//     Enc/Inputs/In/nState1 @bit 4 <-> ENC Status compact/Status/Counter overflow
//     Enc/Inputs/In/nState1 @bit 3 <-> ENC Status compact/Status/Counter underflow
//     Enc/Inputs/In/nState1 @bit 7 <-> ENC Status compact/Status/Extrapolation stall
//     Enc/Inputs/In/nState1 <-> ENC Status compact/Status/Latch C valid
//     Enc/Inputs/In/nState1 @bit 1 <-> ENC Status compact/Status/Latch extern valid
//     Enc/Inputs/In/nState1 @bit 2 <-> ENC Status compact/Status/Set counter done
//     Enc/Inputs/In/nState2 @bit 4 <-> ENC Status compact/Status/Status of extern latch
//     Enc/Inputs/In/nState2 <-> ENC Status compact/Status/Status of input A
//     Enc/Inputs/In/nState2 @bit 1 <-> ENC Status compact/Status/Status of input B
//     Enc/Inputs/In/nState2 @bit 2 <-> ENC Status compact/Status/Status of input C
//     Enc/Inputs/In/nState2 @bit 5 <-> ENC Status compact/Status/Sync error
//     Enc/Inputs/In/nState2 @bit 7 <-> ENC Status compact/Status/TxPDO Toggle
//     Enc/Inputs/In/nState4 @bit 1 <-> WcState/InputToggle
//     Enc/Inputs/In/nState4 <-> WcState/WcState
//     Enc/Outputs/Out/nCtrl1 <-> ENC Control compact/Control/Enable latch C
//     Enc/Outputs/Out/nCtrl1 @bit 3 <-> ENC Control compact/Control/Enable latch extern on negative edge
//     Enc/Outputs/Out/nCtrl1 @bit 1 <-> ENC Control compact/Control/Enable latch extern on positive edge
//     Enc/Outputs/Out/nCtrl1 @bit 2 <-> ENC Control compact/Control/Set counter
//     Enc/Outputs/Out/nDataOut1[0] <-> ENC Control compact/Set counter value
//   NC-Task 1 SAF/Axes/NSH4 <-> Device 1 (EtherCAT)/Term 7 (EK1101)/Term 14 (EK1122)/Term 15 (EK1101)/NSH4 (N19) (EL7047)
//     Drive/Inputs/In/nState1 @bit 3 <-> STM Status/Status/Error
//     Drive/Inputs/In/nState1 @bit 7 <-> STM Status/Status/Motor stall
//     Drive/Inputs/In/nState1 @bit 5 <-> STM Status/Status/Moving negative
//     Drive/Inputs/In/nState1 @bit 4 <-> STM Status/Status/Moving positive
//     Drive/Inputs/In/nState1 @bit 1 <-> STM Status/Status/Ready
//     Drive/Inputs/In/nState1 <-> STM Status/Status/Ready to enable
//     Drive/Inputs/In/nState1 @bit 6 <-> STM Status/Status/Torque reduced
//     Drive/Inputs/In/nState1 @bit 2 <-> STM Status/Status/Warning
//     Drive/Inputs/In/nState2 @bit 3 <-> STM Status/Status/Digital input 1
//     Drive/Inputs/In/nState2 @bit 4 <-> STM Status/Status/Digital input 2
//     Drive/Inputs/In/nState2 @bit 5 <-> STM Status/Status/Sync error
//     Drive/Inputs/In/nState2 @bit 7 <-> STM Status/Status/TxPDO Toggle
//     Drive/Inputs/In/nState4 @bit 1 <-> WcState/InputToggle
//     Drive/Inputs/In/nState4 <-> WcState/WcState
//     Drive/Outputs/Out/nCtrl1 <-> STM Control/Control/Enable
//     Drive/Outputs/Out/nCtrl1 @bit 2 <-> STM Control/Control/Reduce torque
//     Drive/Outputs/Out/nCtrl1 @bit 1 <-> STM Control/Control/Reset
//     Drive/Outputs/Out/nCtrl2 @bit 3 <-> STM Control/Control/Digital output 1
//     Drive/Outputs/Out/nDataOut2[0] <-> STM Velocity/Velocity
//     Enc/Inputs/In/nDataIn1[0] <-> ENC Status compact/Counter value
//     Enc/Inputs/In/nDataIn2[0] <-> ENC Status compact/Latch value
//     Enc/Inputs/In/nState1 @bit 4 <-> ENC Status compact/Status/Counter overflow
//     Enc/Inputs/In/nState1 @bit 3 <-> ENC Status compact/Status/Counter underflow
//     Enc/Inputs/In/nState1 @bit 7 <-> ENC Status compact/Status/Extrapolation stall
//     Enc/Inputs/In/nState1 <-> ENC Status compact/Status/Latch C valid
//     Enc/Inputs/In/nState1 @bit 1 <-> ENC Status compact/Status/Latch extern valid
//     Enc/Inputs/In/nState1 @bit 2 <-> ENC Status compact/Status/Set counter done
//     Enc/Inputs/In/nState2 @bit 4 <-> ENC Status compact/Status/Status of extern latch
//     Enc/Inputs/In/nState2 <-> ENC Status compact/Status/Status of input A
//     Enc/Inputs/In/nState2 @bit 1 <-> ENC Status compact/Status/Status of input B
//     Enc/Inputs/In/nState2 @bit 2 <-> ENC Status compact/Status/Status of input C
//     Enc/Inputs/In/nState2 @bit 5 <-> ENC Status compact/Status/Sync error
//     Enc/Inputs/In/nState2 @bit 7 <-> ENC Status compact/Status/TxPDO Toggle
//     Enc/Inputs/In/nState4 @bit 1 <-> WcState/InputToggle
//     Enc/Inputs/In/nState4 <-> WcState/WcState
//     Enc/Outputs/Out/nCtrl1 <-> ENC Control compact/Control/Enable latch C
//     Enc/Outputs/Out/nCtrl1 @bit 3 <-> ENC Control compact/Control/Enable latch extern on negative edge
//     Enc/Outputs/Out/nCtrl1 @bit 1 <-> ENC Control compact/Control/Enable latch extern on positive edge
//     Enc/Outputs/Out/nCtrl1 @bit 2 <-> ENC Control compact/Control/Set counter
//     Enc/Outputs/Out/nDataOut1[0] <-> ENC Control compact/Set counter value
//   NC-Task 1 SAF/Axes/NTPA1 <-> Device 1 (EtherCAT)/Term 7 (EK1101)/Term 14 (EK1122)/Term 32 (EK1101)/NTPA1 - NTPA2 (N6) (EL7342)
//     Drive/Inputs/In/nState1 @bit 3 <-> DCM Status Channel 1/Status/Error
//     Drive/Inputs/In/nState1 @bit 5 <-> DCM Status Channel 1/Status/Moving negative
//     Drive/Inputs/In/nState1 @bit 4 <-> DCM Status Channel 1/Status/Moving positive
//     Drive/Inputs/In/nState1 @bit 1 <-> DCM Status Channel 1/Status/Ready
//     Drive/Inputs/In/nState1 <-> DCM Status Channel 1/Status/Ready to enable
//     Drive/Inputs/In/nState1 @bit 6 <-> DCM Status Channel 1/Status/Torque reduced
//     Drive/Inputs/In/nState1 @bit 2 <-> DCM Status Channel 1/Status/Warning
//     Drive/Inputs/In/nState2 @bit 3 <-> DCM Status Channel 1/Status/Digital input 1
//     Drive/Inputs/In/nState2 @bit 4 <-> DCM Status Channel 1/Status/Digital input 2
//     Drive/Inputs/In/nState2 @bit 5 <-> DCM Status Channel 1/Status/Sync error
//     Drive/Inputs/In/nState2 @bit 7 <-> DCM Status Channel 1/Status/TxPDO Toggle
//     Drive/Inputs/In/nState4 @bit 1 <-> WcState/InputToggle
//     Drive/Inputs/In/nState4 <-> WcState/WcState
//     Drive/Outputs/Out/nCtrl1 <-> DCM Control Channel 1/Control/Enable
//     Drive/Outputs/Out/nCtrl1 @bit 2 <-> DCM Control Channel 1/Control/Reduce torque
//     Drive/Outputs/Out/nCtrl1 @bit 1 <-> DCM Control Channel 1/Control/Reset
//     Drive/Outputs/Out/nCtrl1 @bit 3 <-> DCM Control Channel 1/Control/Threshold active
//     Drive/Outputs/Out/nDataOut2[0] <-> DCM Velocity Channel 1/Velocity
//     Enc/Inputs/In/nDataIn1[0] <-> ENC Status compact Channel 1/Counter value
//     Enc/Inputs/In/nDataIn2[0] <-> ENC Status compact Channel 1/Latch value
//     Enc/Inputs/In/nState1 @bit 4 <-> ENC Status compact Channel 1/Status/Counter overflow
//     Enc/Inputs/In/nState1 @bit 3 <-> ENC Status compact Channel 1/Status/Counter underflow
//     Enc/Inputs/In/nState1 @bit 7 <-> ENC Status compact Channel 1/Status/Extrapolation stall
//     Enc/Inputs/In/nState1 @bit 1 <-> ENC Status compact Channel 1/Status/Latch extern valid
//     Enc/Inputs/In/nState1 @bit 2 <-> ENC Status compact Channel 1/Status/Set counter done
//     Enc/Inputs/In/nState2 @bit 4 <-> ENC Status compact Channel 1/Status/Status of extern latch
//     Enc/Inputs/In/nState2 <-> ENC Status compact Channel 1/Status/Status of input A
//     Enc/Inputs/In/nState2 @bit 1 <-> ENC Status compact Channel 1/Status/Status of input B
//     Enc/Inputs/In/nState2 @bit 5 <-> ENC Status compact Channel 1/Status/Sync error
//     Enc/Inputs/In/nState2 @bit 7 <-> ENC Status compact Channel 1/Status/TxPDO Toggle
//     Enc/Inputs/In/nState4 @bit 1 <-> WcState/InputToggle
//     Enc/Inputs/In/nState4 <-> WcState/WcState
//     Enc/Outputs/Out/nCtrl1 @bit 3 <-> ENC Control compact Channel 1/Control/Enable latch extern on negative edge
//     Enc/Outputs/Out/nCtrl1 @bit 1 <-> ENC Control compact Channel 1/Control/Enable latch extern on positive edge
//     Enc/Outputs/Out/nCtrl1 @bit 2 <-> ENC Control compact Channel 1/Control/Set counter
//     Enc/Outputs/Out/nDataOut1[0] <-> ENC Control compact Channel 1/Set counter value
//   NC-Task 1 SAF/Axes/NTPA2 <-> Device 1 (EtherCAT)/Term 7 (EK1101)/Term 14 (EK1122)/Term 32 (EK1101)/NTPA1 - NTPA2 (N6) (EL7342)
//     Drive/Inputs/In/nState1 @bit 3 <-> DCM Status Channel 2/Status/Error
//     Drive/Inputs/In/nState1 @bit 5 <-> DCM Status Channel 2/Status/Moving negative
//     Drive/Inputs/In/nState1 @bit 4 <-> DCM Status Channel 2/Status/Moving positive
//     Drive/Inputs/In/nState1 @bit 1 <-> DCM Status Channel 2/Status/Ready
//     Drive/Inputs/In/nState1 <-> DCM Status Channel 2/Status/Ready to enable
//     Drive/Inputs/In/nState1 @bit 6 <-> DCM Status Channel 2/Status/Torque reduced
//     Drive/Inputs/In/nState1 @bit 2 <-> DCM Status Channel 2/Status/Warning
//     Drive/Inputs/In/nState2 @bit 3 <-> DCM Status Channel 2/Status/Digital input 1
//     Drive/Inputs/In/nState2 @bit 4 <-> DCM Status Channel 2/Status/Digital input 2
//     Drive/Inputs/In/nState2 @bit 5 <-> DCM Status Channel 2/Status/Sync error
//     Drive/Inputs/In/nState2 @bit 7 <-> DCM Status Channel 2/Status/TxPDO Toggle
//     Drive/Inputs/In/nState4 @bit 1 <-> WcState/InputToggle
//     Drive/Inputs/In/nState4 <-> WcState/WcState
//     Drive/Outputs/Out/nCtrl1 <-> DCM Control Channel 2/Control/Enable
//     Drive/Outputs/Out/nCtrl1 @bit 2 <-> DCM Control Channel 2/Control/Reduce torque
//     Drive/Outputs/Out/nCtrl1 @bit 1 <-> DCM Control Channel 2/Control/Reset
//     Drive/Outputs/Out/nCtrl1 @bit 3 <-> DCM Control Channel 2/Control/Threshold active
//     Drive/Outputs/Out/nDataOut2[0] <-> DCM Velocity Channel 2/Velocity
//     Enc/Inputs/In/nDataIn1[0] <-> ENC Status compact Channel 2/Counter value
//     Enc/Inputs/In/nDataIn2[0] <-> ENC Status compact Channel 2/Latch value
//     Enc/Inputs/In/nState1 @bit 4 <-> ENC Status compact Channel 2/Status/Counter overflow
//     Enc/Inputs/In/nState1 @bit 3 <-> ENC Status compact Channel 2/Status/Counter underflow
//     Enc/Inputs/In/nState1 @bit 7 <-> ENC Status compact Channel 2/Status/Extrapolation stall
//     Enc/Inputs/In/nState1 @bit 1 <-> ENC Status compact Channel 2/Status/Latch extern valid
//     Enc/Inputs/In/nState1 @bit 2 <-> ENC Status compact Channel 2/Status/Set counter done
//     Enc/Inputs/In/nState2 @bit 4 <-> ENC Status compact Channel 2/Status/Status of extern latch
//     Enc/Inputs/In/nState2 <-> ENC Status compact Channel 2/Status/Status of input A
//     Enc/Inputs/In/nState2 @bit 1 <-> ENC Status compact Channel 2/Status/Status of input B
//     Enc/Inputs/In/nState2 @bit 5 <-> ENC Status compact Channel 2/Status/Sync error
//     Enc/Inputs/In/nState2 @bit 7 <-> ENC Status compact Channel 2/Status/TxPDO Toggle
//     Enc/Inputs/In/nState4 @bit 1 <-> WcState/InputToggle
//     Enc/Inputs/In/nState4 <-> WcState/WcState
//     Enc/Outputs/Out/nCtrl1 @bit 3 <-> ENC Control compact Channel 2/Control/Enable latch extern on negative edge
//     Enc/Outputs/Out/nCtrl1 @bit 1 <-> ENC Control compact Channel 2/Control/Enable latch extern on positive edge
//     Enc/Outputs/Out/nCtrl1 @bit 2 <-> ENC Control compact Channel 2/Control/Set counter
//     Enc/Outputs/Out/nDataOut1[0] <-> ENC Control compact Channel 2/Set counter value
//   NC-Task 1 SAF/Axes/NTPA3 <-> Device 1 (EtherCAT)/Term 7 (EK1101)/Term 14 (EK1122)/Term 32 (EK1101)/NTPA3 - NTPA4 (N7) (EL7342)
//     Drive/Inputs/In/nState1 @bit 3 <-> DCM Status Channel 1/Status/Error
//     Drive/Inputs/In/nState1 @bit 5 <-> DCM Status Channel 1/Status/Moving negative
//     Drive/Inputs/In/nState1 @bit 4 <-> DCM Status Channel 1/Status/Moving positive
//     Drive/Inputs/In/nState1 @bit 1 <-> DCM Status Channel 1/Status/Ready
//     Drive/Inputs/In/nState1 <-> DCM Status Channel 1/Status/Ready to enable
//     Drive/Inputs/In/nState1 @bit 6 <-> DCM Status Channel 1/Status/Torque reduced
//     Drive/Inputs/In/nState1 @bit 2 <-> DCM Status Channel 1/Status/Warning
//     Drive/Inputs/In/nState2 @bit 3 <-> DCM Status Channel 1/Status/Digital input 1
//     Drive/Inputs/In/nState2 @bit 4 <-> DCM Status Channel 1/Status/Digital input 2
//     Drive/Inputs/In/nState2 @bit 5 <-> DCM Status Channel 1/Status/Sync error
//     Drive/Inputs/In/nState2 @bit 7 <-> DCM Status Channel 1/Status/TxPDO Toggle
//     Drive/Inputs/In/nState4 @bit 1 <-> WcState/InputToggle
//     Drive/Inputs/In/nState4 <-> WcState/WcState
//     Drive/Outputs/Out/nCtrl1 <-> DCM Control Channel 1/Control/Enable
//     Drive/Outputs/Out/nCtrl1 @bit 2 <-> DCM Control Channel 1/Control/Reduce torque
//     Drive/Outputs/Out/nCtrl1 @bit 1 <-> DCM Control Channel 1/Control/Reset
//     Drive/Outputs/Out/nCtrl1 @bit 3 <-> DCM Control Channel 1/Control/Threshold active
//     Drive/Outputs/Out/nDataOut2[0] <-> DCM Velocity Channel 1/Velocity
//     Enc/Inputs/In/nDataIn1[0] <-> ENC Status compact Channel 1/Counter value
//     Enc/Inputs/In/nDataIn2[0] <-> ENC Status compact Channel 1/Latch value
//     Enc/Inputs/In/nState1 @bit 4 <-> ENC Status compact Channel 1/Status/Counter overflow
//     Enc/Inputs/In/nState1 @bit 3 <-> ENC Status compact Channel 1/Status/Counter underflow
//     Enc/Inputs/In/nState1 @bit 7 <-> ENC Status compact Channel 1/Status/Extrapolation stall
//     Enc/Inputs/In/nState1 @bit 1 <-> ENC Status compact Channel 1/Status/Latch extern valid
//     Enc/Inputs/In/nState1 @bit 2 <-> ENC Status compact Channel 1/Status/Set counter done
//     Enc/Inputs/In/nState2 @bit 4 <-> ENC Status compact Channel 1/Status/Status of extern latch
//     Enc/Inputs/In/nState2 <-> ENC Status compact Channel 1/Status/Status of input A
//     Enc/Inputs/In/nState2 @bit 1 <-> ENC Status compact Channel 1/Status/Status of input B
//     Enc/Inputs/In/nState2 @bit 5 <-> ENC Status compact Channel 1/Status/Sync error
//     Enc/Inputs/In/nState2 @bit 7 <-> ENC Status compact Channel 1/Status/TxPDO Toggle
//     Enc/Inputs/In/nState4 @bit 1 <-> WcState/InputToggle
//     Enc/Inputs/In/nState4 <-> WcState/WcState
//     Enc/Outputs/Out/nCtrl1 @bit 3 <-> ENC Control compact Channel 1/Control/Enable latch extern on negative edge
//     Enc/Outputs/Out/nCtrl1 @bit 1 <-> ENC Control compact Channel 1/Control/Enable latch extern on positive edge
//     Enc/Outputs/Out/nCtrl1 @bit 2 <-> ENC Control compact Channel 1/Control/Set counter
//     Enc/Outputs/Out/nDataOut1[0] <-> ENC Control compact Channel 1/Set counter value
//   NC-Task 1 SAF/Axes/NTPA4 <-> Device 1 (EtherCAT)/Term 7 (EK1101)/Term 14 (EK1122)/Term 32 (EK1101)/NTPA3 - NTPA4 (N7) (EL7342)
//     Drive/Inputs/In/nState1 @bit 3 <-> DCM Status Channel 2/Status/Error
//     Drive/Inputs/In/nState1 @bit 5 <-> DCM Status Channel 2/Status/Moving negative
//     Drive/Inputs/In/nState1 @bit 4 <-> DCM Status Channel 2/Status/Moving positive
//     Drive/Inputs/In/nState1 @bit 1 <-> DCM Status Channel 2/Status/Ready
//     Drive/Inputs/In/nState1 <-> DCM Status Channel 2/Status/Ready to enable
//     Drive/Inputs/In/nState1 @bit 6 <-> DCM Status Channel 2/Status/Torque reduced
//     Drive/Inputs/In/nState1 @bit 2 <-> DCM Status Channel 2/Status/Warning
//     Drive/Inputs/In/nState2 @bit 3 <-> DCM Status Channel 2/Status/Digital input 1
//     Drive/Inputs/In/nState2 @bit 4 <-> DCM Status Channel 2/Status/Digital input 2
//     Drive/Inputs/In/nState2 @bit 5 <-> DCM Status Channel 2/Status/Sync error
//     Drive/Inputs/In/nState2 @bit 7 <-> DCM Status Channel 2/Status/TxPDO Toggle
//     Drive/Inputs/In/nState4 @bit 1 <-> WcState/InputToggle
//     Drive/Inputs/In/nState4 <-> WcState/WcState
//     Drive/Outputs/Out/nCtrl1 <-> DCM Control Channel 2/Control/Enable
//     Drive/Outputs/Out/nCtrl1 @bit 2 <-> DCM Control Channel 2/Control/Reduce torque
//     Drive/Outputs/Out/nCtrl1 @bit 1 <-> DCM Control Channel 2/Control/Reset
//     Drive/Outputs/Out/nCtrl1 @bit 3 <-> DCM Control Channel 2/Control/Threshold active
//     Drive/Outputs/Out/nDataOut2[0] <-> DCM Velocity Channel 2/Velocity
//     Enc/Inputs/In/nDataIn1[0] <-> ENC Status compact Channel 2/Counter value
//     Enc/Inputs/In/nDataIn2[0] <-> ENC Status compact Channel 2/Latch value
//     Enc/Inputs/In/nState1 @bit 4 <-> ENC Status compact Channel 2/Status/Counter overflow
//     Enc/Inputs/In/nState1 @bit 3 <-> ENC Status compact Channel 2/Status/Counter underflow
//     Enc/Inputs/In/nState1 @bit 7 <-> ENC Status compact Channel 2/Status/Extrapolation stall
//     Enc/Inputs/In/nState1 @bit 1 <-> ENC Status compact Channel 2/Status/Latch extern valid
//     Enc/Inputs/In/nState1 @bit 2 <-> ENC Status compact Channel 2/Status/Set counter done
//     Enc/Inputs/In/nState2 @bit 4 <-> ENC Status compact Channel 2/Status/Status of extern latch
//     Enc/Inputs/In/nState2 <-> ENC Status compact Channel 2/Status/Status of input A
//     Enc/Inputs/In/nState2 @bit 1 <-> ENC Status compact Channel 2/Status/Status of input B
//     Enc/Inputs/In/nState2 @bit 5 <-> ENC Status compact Channel 2/Status/Sync error
//     Enc/Inputs/In/nState2 @bit 7 <-> ENC Status compact Channel 2/Status/TxPDO Toggle
//     Enc/Inputs/In/nState4 @bit 1 <-> WcState/InputToggle
//     Enc/Inputs/In/nState4 <-> WcState/WcState
//     Enc/Outputs/Out/nCtrl1 @bit 3 <-> ENC Control compact Channel 2/Control/Enable latch extern on negative edge
//     Enc/Outputs/Out/nCtrl1 @bit 1 <-> ENC Control compact Channel 2/Control/Enable latch extern on positive edge
//     Enc/Outputs/Out/nCtrl1 @bit 2 <-> ENC Control compact Channel 2/Control/Set counter
//     Enc/Outputs/Out/nDataOut1[0] <-> ENC Control compact Channel 2/Set counter value
//   NC-Task 1 SAF/Axes/NTPB1 <-> Device 1 (EtherCAT)/Term 7 (EK1101)/Term 14 (EK1122)/Term 32 (EK1101)/NTPB1 - NTPB2 (N14) (EL7342)
//     Drive/Inputs/In/nState1 @bit 3 <-> DCM Status Channel 1/Status/Error
//     Drive/Inputs/In/nState1 @bit 5 <-> DCM Status Channel 1/Status/Moving negative
//     Drive/Inputs/In/nState1 @bit 4 <-> DCM Status Channel 1/Status/Moving positive
//     Drive/Inputs/In/nState1 @bit 1 <-> DCM Status Channel 1/Status/Ready
//     Drive/Inputs/In/nState1 <-> DCM Status Channel 1/Status/Ready to enable
//     Drive/Inputs/In/nState1 @bit 6 <-> DCM Status Channel 1/Status/Torque reduced
//     Drive/Inputs/In/nState1 @bit 2 <-> DCM Status Channel 1/Status/Warning
//     Drive/Inputs/In/nState2 @bit 3 <-> DCM Status Channel 1/Status/Digital input 1
//     Drive/Inputs/In/nState2 @bit 4 <-> DCM Status Channel 1/Status/Digital input 2
//     Drive/Inputs/In/nState2 @bit 5 <-> DCM Status Channel 1/Status/Sync error
//     Drive/Inputs/In/nState2 @bit 7 <-> DCM Status Channel 1/Status/TxPDO Toggle
//     Drive/Inputs/In/nState4 @bit 1 <-> WcState/InputToggle
//     Drive/Inputs/In/nState4 <-> WcState/WcState
//     Drive/Outputs/Out/nCtrl1 <-> DCM Control Channel 1/Control/Enable
//     Drive/Outputs/Out/nCtrl1 @bit 2 <-> DCM Control Channel 1/Control/Reduce torque
//     Drive/Outputs/Out/nCtrl1 @bit 1 <-> DCM Control Channel 1/Control/Reset
//     Drive/Outputs/Out/nCtrl1 @bit 3 <-> DCM Control Channel 1/Control/Threshold active
//     Drive/Outputs/Out/nDataOut2[0] <-> DCM Velocity Channel 1/Velocity
//     Enc/Inputs/In/nDataIn1[0] <-> ENC Status compact Channel 1/Counter value
//     Enc/Inputs/In/nDataIn2[0] <-> ENC Status compact Channel 1/Latch value
//     Enc/Inputs/In/nState1 @bit 4 <-> ENC Status compact Channel 1/Status/Counter overflow
//     Enc/Inputs/In/nState1 @bit 3 <-> ENC Status compact Channel 1/Status/Counter underflow
//     Enc/Inputs/In/nState1 @bit 7 <-> ENC Status compact Channel 1/Status/Extrapolation stall
//     Enc/Inputs/In/nState1 @bit 1 <-> ENC Status compact Channel 1/Status/Latch extern valid
//     Enc/Inputs/In/nState1 @bit 2 <-> ENC Status compact Channel 1/Status/Set counter done
//     Enc/Inputs/In/nState2 @bit 4 <-> ENC Status compact Channel 1/Status/Status of extern latch
//     Enc/Inputs/In/nState2 <-> ENC Status compact Channel 1/Status/Status of input A
//     Enc/Inputs/In/nState2 @bit 1 <-> ENC Status compact Channel 1/Status/Status of input B
//     Enc/Inputs/In/nState2 @bit 5 <-> ENC Status compact Channel 1/Status/Sync error
//     Enc/Inputs/In/nState2 @bit 7 <-> ENC Status compact Channel 1/Status/TxPDO Toggle
//     Enc/Inputs/In/nState4 @bit 1 <-> WcState/InputToggle
//     Enc/Inputs/In/nState4 <-> WcState/WcState
//     Enc/Outputs/Out/nCtrl1 @bit 3 <-> ENC Control compact Channel 1/Control/Enable latch extern on negative edge
//     Enc/Outputs/Out/nCtrl1 @bit 1 <-> ENC Control compact Channel 1/Control/Enable latch extern on positive edge
//     Enc/Outputs/Out/nCtrl1 @bit 2 <-> ENC Control compact Channel 1/Control/Set counter
//     Enc/Outputs/Out/nDataOut1[0] <-> ENC Control compact Channel 1/Set counter value
//   NC-Task 1 SAF/Axes/NTPB2 <-> Device 1 (EtherCAT)/Term 7 (EK1101)/Term 14 (EK1122)/Term 32 (EK1101)/NTPB1 - NTPB2 (N14) (EL7342)
//     Drive/Inputs/In/nState1 @bit 3 <-> DCM Status Channel 2/Status/Error
//     Drive/Inputs/In/nState1 @bit 5 <-> DCM Status Channel 2/Status/Moving negative
//     Drive/Inputs/In/nState1 @bit 4 <-> DCM Status Channel 2/Status/Moving positive
//     Drive/Inputs/In/nState1 @bit 1 <-> DCM Status Channel 2/Status/Ready
//     Drive/Inputs/In/nState1 <-> DCM Status Channel 2/Status/Ready to enable
//     Drive/Inputs/In/nState1 @bit 6 <-> DCM Status Channel 2/Status/Torque reduced
//     Drive/Inputs/In/nState1 @bit 2 <-> DCM Status Channel 2/Status/Warning
//     Drive/Inputs/In/nState2 @bit 3 <-> DCM Status Channel 2/Status/Digital input 1
//     Drive/Inputs/In/nState2 @bit 4 <-> DCM Status Channel 2/Status/Digital input 2
//     Drive/Inputs/In/nState2 @bit 5 <-> DCM Status Channel 2/Status/Sync error
//     Drive/Inputs/In/nState2 @bit 7 <-> DCM Status Channel 2/Status/TxPDO Toggle
//     Drive/Inputs/In/nState4 @bit 1 <-> WcState/InputToggle
//     Drive/Inputs/In/nState4 <-> WcState/WcState
//     Drive/Outputs/Out/nCtrl1 <-> DCM Control Channel 2/Control/Enable
//     Drive/Outputs/Out/nCtrl1 @bit 2 <-> DCM Control Channel 2/Control/Reduce torque
//     Drive/Outputs/Out/nCtrl1 @bit 1 <-> DCM Control Channel 2/Control/Reset
//     Drive/Outputs/Out/nCtrl1 @bit 3 <-> DCM Control Channel 2/Control/Threshold active
//     Drive/Outputs/Out/nDataOut2[0] <-> DCM Velocity Channel 2/Velocity
//     Enc/Inputs/In/nDataIn1[0] <-> ENC Status compact Channel 2/Counter value
//     Enc/Inputs/In/nDataIn2[0] <-> ENC Status compact Channel 2/Latch value
//     Enc/Inputs/In/nState1 @bit 4 <-> ENC Status compact Channel 2/Status/Counter overflow
//     Enc/Inputs/In/nState1 @bit 3 <-> ENC Status compact Channel 2/Status/Counter underflow
//     Enc/Inputs/In/nState1 @bit 7 <-> ENC Status compact Channel 2/Status/Extrapolation stall
//     Enc/Inputs/In/nState1 @bit 1 <-> ENC Status compact Channel 2/Status/Latch extern valid
//     Enc/Inputs/In/nState1 @bit 2 <-> ENC Status compact Channel 2/Status/Set counter done
//     Enc/Inputs/In/nState2 @bit 4 <-> ENC Status compact Channel 2/Status/Status of extern latch
//     Enc/Inputs/In/nState2 <-> ENC Status compact Channel 2/Status/Status of input A
//     Enc/Inputs/In/nState2 @bit 1 <-> ENC Status compact Channel 2/Status/Status of input B
//     Enc/Inputs/In/nState2 @bit 5 <-> ENC Status compact Channel 2/Status/Sync error
//     Enc/Inputs/In/nState2 @bit 7 <-> ENC Status compact Channel 2/Status/TxPDO Toggle
//     Enc/Inputs/In/nState4 @bit 1 <-> WcState/InputToggle
//     Enc/Inputs/In/nState4 <-> WcState/WcState
//     Enc/Outputs/Out/nCtrl1 @bit 3 <-> ENC Control compact Channel 2/Control/Enable latch extern on negative edge
//     Enc/Outputs/Out/nCtrl1 @bit 1 <-> ENC Control compact Channel 2/Control/Enable latch extern on positive edge
//     Enc/Outputs/Out/nCtrl1 @bit 2 <-> ENC Control compact Channel 2/Control/Set counter
//     Enc/Outputs/Out/nDataOut1[0] <-> ENC Control compact Channel 2/Set counter value
//   NC-Task 1 SAF/Axes/NTPB3 <-> Device 1 (EtherCAT)/Term 7 (EK1101)/Term 14 (EK1122)/Term 32 (EK1101)/NTPB3 - NTPB4 (N15) (EL7342)
//     Drive/Inputs/In/nState1 @bit 3 <-> DCM Status Channel 1/Status/Error
//     Drive/Inputs/In/nState1 @bit 5 <-> DCM Status Channel 1/Status/Moving negative
//     Drive/Inputs/In/nState1 @bit 4 <-> DCM Status Channel 1/Status/Moving positive
//     Drive/Inputs/In/nState1 @bit 1 <-> DCM Status Channel 1/Status/Ready
//     Drive/Inputs/In/nState1 <-> DCM Status Channel 1/Status/Ready to enable
//     Drive/Inputs/In/nState1 @bit 6 <-> DCM Status Channel 1/Status/Torque reduced
//     Drive/Inputs/In/nState1 @bit 2 <-> DCM Status Channel 1/Status/Warning
//     Drive/Inputs/In/nState2 @bit 3 <-> DCM Status Channel 1/Status/Digital input 1
//     Drive/Inputs/In/nState2 @bit 4 <-> DCM Status Channel 1/Status/Digital input 2
//     Drive/Inputs/In/nState2 @bit 5 <-> DCM Status Channel 1/Status/Sync error
//     Drive/Inputs/In/nState2 @bit 7 <-> DCM Status Channel 1/Status/TxPDO Toggle
//     Drive/Inputs/In/nState4 @bit 1 <-> WcState/InputToggle
//     Drive/Inputs/In/nState4 <-> WcState/WcState
//     Drive/Outputs/Out/nCtrl1 <-> DCM Control Channel 1/Control/Enable
//     Drive/Outputs/Out/nCtrl1 @bit 2 <-> DCM Control Channel 1/Control/Reduce torque
//     Drive/Outputs/Out/nCtrl1 @bit 1 <-> DCM Control Channel 1/Control/Reset
//     Drive/Outputs/Out/nCtrl1 @bit 3 <-> DCM Control Channel 1/Control/Threshold active
//     Drive/Outputs/Out/nDataOut2[0] <-> DCM Velocity Channel 1/Velocity
//     Enc/Inputs/In/nDataIn1[0] <-> ENC Status compact Channel 1/Counter value
//     Enc/Inputs/In/nDataIn2[0] <-> ENC Status compact Channel 1/Latch value
//     Enc/Inputs/In/nState1 @bit 4 <-> ENC Status compact Channel 1/Status/Counter overflow
//     Enc/Inputs/In/nState1 @bit 3 <-> ENC Status compact Channel 1/Status/Counter underflow
//     Enc/Inputs/In/nState1 @bit 7 <-> ENC Status compact Channel 1/Status/Extrapolation stall
//     Enc/Inputs/In/nState1 @bit 1 <-> ENC Status compact Channel 1/Status/Latch extern valid
//     Enc/Inputs/In/nState1 @bit 2 <-> ENC Status compact Channel 1/Status/Set counter done
//     Enc/Inputs/In/nState2 @bit 4 <-> ENC Status compact Channel 1/Status/Status of extern latch
//     Enc/Inputs/In/nState2 <-> ENC Status compact Channel 1/Status/Status of input A
//     Enc/Inputs/In/nState2 @bit 1 <-> ENC Status compact Channel 1/Status/Status of input B
//     Enc/Inputs/In/nState2 @bit 5 <-> ENC Status compact Channel 1/Status/Sync error
//     Enc/Inputs/In/nState2 @bit 7 <-> ENC Status compact Channel 1/Status/TxPDO Toggle
//     Enc/Inputs/In/nState4 @bit 1 <-> WcState/InputToggle
//     Enc/Inputs/In/nState4 <-> WcState/WcState
//     Enc/Outputs/Out/nCtrl1 @bit 3 <-> ENC Control compact Channel 1/Control/Enable latch extern on negative edge
//     Enc/Outputs/Out/nCtrl1 @bit 1 <-> ENC Control compact Channel 1/Control/Enable latch extern on positive edge
//     Enc/Outputs/Out/nCtrl1 @bit 2 <-> ENC Control compact Channel 1/Control/Set counter
//     Enc/Outputs/Out/nDataOut1[0] <-> ENC Control compact Channel 1/Set counter value
//   NC-Task 1 SAF/Axes/NTPB4 <-> Device 1 (EtherCAT)/Term 7 (EK1101)/Term 14 (EK1122)/Term 32 (EK1101)/NTPB3 - NTPB4 (N15) (EL7342)
//     Drive/Inputs/In/nState1 @bit 3 <-> DCM Status Channel 2/Status/Error
//     Drive/Inputs/In/nState1 @bit 5 <-> DCM Status Channel 2/Status/Moving negative
//     Drive/Inputs/In/nState1 @bit 4 <-> DCM Status Channel 2/Status/Moving positive
//     Drive/Inputs/In/nState1 @bit 1 <-> DCM Status Channel 2/Status/Ready
//     Drive/Inputs/In/nState1 <-> DCM Status Channel 2/Status/Ready to enable
//     Drive/Inputs/In/nState1 @bit 6 <-> DCM Status Channel 2/Status/Torque reduced
//     Drive/Inputs/In/nState1 @bit 2 <-> DCM Status Channel 2/Status/Warning
//     Drive/Inputs/In/nState2 @bit 3 <-> DCM Status Channel 2/Status/Digital input 1
//     Drive/Inputs/In/nState2 @bit 4 <-> DCM Status Channel 2/Status/Digital input 2
//     Drive/Inputs/In/nState2 @bit 5 <-> DCM Status Channel 2/Status/Sync error
//     Drive/Inputs/In/nState2 @bit 7 <-> DCM Status Channel 2/Status/TxPDO Toggle
//     Drive/Inputs/In/nState4 @bit 1 <-> WcState/InputToggle
//     Drive/Inputs/In/nState4 <-> WcState/WcState
//     Drive/Outputs/Out/nCtrl1 <-> DCM Control Channel 2/Control/Enable
//     Drive/Outputs/Out/nCtrl1 @bit 2 <-> DCM Control Channel 2/Control/Reduce torque
//     Drive/Outputs/Out/nCtrl1 @bit 1 <-> DCM Control Channel 2/Control/Reset
//     Drive/Outputs/Out/nCtrl1 @bit 3 <-> DCM Control Channel 2/Control/Threshold active
//     Drive/Outputs/Out/nDataOut2[0] <-> DCM Velocity Channel 2/Velocity
//     Enc/Inputs/In/nDataIn1[0] <-> ENC Status compact Channel 2/Counter value
//     Enc/Inputs/In/nDataIn2[0] <-> ENC Status compact Channel 2/Latch value
//     Enc/Inputs/In/nState1 @bit 4 <-> ENC Status compact Channel 2/Status/Counter overflow
//     Enc/Inputs/In/nState1 @bit 3 <-> ENC Status compact Channel 2/Status/Counter underflow
//     Enc/Inputs/In/nState1 @bit 7 <-> ENC Status compact Channel 2/Status/Extrapolation stall
//     Enc/Inputs/In/nState1 @bit 1 <-> ENC Status compact Channel 2/Status/Latch extern valid
//     Enc/Inputs/In/nState1 @bit 2 <-> ENC Status compact Channel 2/Status/Set counter done
//     Enc/Inputs/In/nState2 @bit 4 <-> ENC Status compact Channel 2/Status/Status of extern latch
//     Enc/Inputs/In/nState2 <-> ENC Status compact Channel 2/Status/Status of input A
//     Enc/Inputs/In/nState2 @bit 1 <-> ENC Status compact Channel 2/Status/Status of input B
//     Enc/Inputs/In/nState2 @bit 5 <-> ENC Status compact Channel 2/Status/Sync error
//     Enc/Inputs/In/nState2 @bit 7 <-> ENC Status compact Channel 2/Status/TxPDO Toggle
//     Enc/Inputs/In/nState4 @bit 1 <-> WcState/InputToggle
//     Enc/Inputs/In/nState4 <-> WcState/WcState
//     Enc/Outputs/Out/nCtrl1 @bit 3 <-> ENC Control compact Channel 2/Control/Enable latch extern on negative edge
//     Enc/Outputs/Out/nCtrl1 @bit 1 <-> ENC Control compact Channel 2/Control/Enable latch extern on positive edge
//     Enc/Outputs/Out/nCtrl1 @bit 2 <-> ENC Control compact Channel 2/Control/Set counter
//     Enc/Outputs/Out/nDataOut1[0] <-> ENC Control compact Channel 2/Set counter value
//   NC-Task 1 SAF/Axes/NTTA1 <-> Device 1 (EtherCAT)/Term 7 (EK1101)/Term 14 (EK1122)/Term 32 (EK1101)/NTTA1 - NTTA2 (N9) (EL7342)
//     Drive/Inputs/In/nState1 @bit 3 <-> DCM Status Channel 1/Status/Error
//     Drive/Inputs/In/nState1 @bit 5 <-> DCM Status Channel 1/Status/Moving negative
//     Drive/Inputs/In/nState1 @bit 4 <-> DCM Status Channel 1/Status/Moving positive
//     Drive/Inputs/In/nState1 @bit 1 <-> DCM Status Channel 1/Status/Ready
//     Drive/Inputs/In/nState1 <-> DCM Status Channel 1/Status/Ready to enable
//     Drive/Inputs/In/nState1 @bit 6 <-> DCM Status Channel 1/Status/Torque reduced
//     Drive/Inputs/In/nState1 @bit 2 <-> DCM Status Channel 1/Status/Warning
//     Drive/Inputs/In/nState2 @bit 3 <-> DCM Status Channel 1/Status/Digital input 1
//     Drive/Inputs/In/nState2 @bit 4 <-> DCM Status Channel 1/Status/Digital input 2
//     Drive/Inputs/In/nState2 @bit 5 <-> DCM Status Channel 1/Status/Sync error
//     Drive/Inputs/In/nState2 @bit 7 <-> DCM Status Channel 1/Status/TxPDO Toggle
//     Drive/Inputs/In/nState4 @bit 1 <-> WcState/InputToggle
//     Drive/Inputs/In/nState4 <-> WcState/WcState
//     Drive/Outputs/Out/nCtrl1 <-> DCM Control Channel 1/Control/Enable
//     Drive/Outputs/Out/nCtrl1 @bit 2 <-> DCM Control Channel 1/Control/Reduce torque
//     Drive/Outputs/Out/nCtrl1 @bit 1 <-> DCM Control Channel 1/Control/Reset
//     Drive/Outputs/Out/nCtrl1 @bit 3 <-> DCM Control Channel 1/Control/Threshold active
//     Drive/Outputs/Out/nDataOut2[0] <-> DCM Velocity Channel 1/Velocity
//     Enc/Inputs/In/nDataIn1[0] <-> ENC Status compact Channel 1/Counter value
//     Enc/Inputs/In/nDataIn2[0] <-> ENC Status compact Channel 1/Latch value
//     Enc/Inputs/In/nState1 @bit 4 <-> ENC Status compact Channel 1/Status/Counter overflow
//     Enc/Inputs/In/nState1 @bit 3 <-> ENC Status compact Channel 1/Status/Counter underflow
//     Enc/Inputs/In/nState1 @bit 7 <-> ENC Status compact Channel 1/Status/Extrapolation stall
//     Enc/Inputs/In/nState1 @bit 1 <-> ENC Status compact Channel 1/Status/Latch extern valid
//     Enc/Inputs/In/nState1 @bit 2 <-> ENC Status compact Channel 1/Status/Set counter done
//     Enc/Inputs/In/nState2 @bit 4 <-> ENC Status compact Channel 1/Status/Status of extern latch
//     Enc/Inputs/In/nState2 <-> ENC Status compact Channel 1/Status/Status of input A
//     Enc/Inputs/In/nState2 @bit 1 <-> ENC Status compact Channel 1/Status/Status of input B
//     Enc/Inputs/In/nState2 @bit 5 <-> ENC Status compact Channel 1/Status/Sync error
//     Enc/Inputs/In/nState2 @bit 7 <-> ENC Status compact Channel 1/Status/TxPDO Toggle
//     Enc/Inputs/In/nState4 @bit 1 <-> WcState/InputToggle
//     Enc/Inputs/In/nState4 <-> WcState/WcState
//     Enc/Outputs/Out/nCtrl1 @bit 3 <-> ENC Control compact Channel 1/Control/Enable latch extern on negative edge
//     Enc/Outputs/Out/nCtrl1 @bit 1 <-> ENC Control compact Channel 1/Control/Enable latch extern on positive edge
//     Enc/Outputs/Out/nCtrl1 @bit 2 <-> ENC Control compact Channel 1/Control/Set counter
//     Enc/Outputs/Out/nDataOut1[0] <-> ENC Control compact Channel 1/Set counter value
//   NC-Task 1 SAF/Axes/NTTA2 <-> Device 1 (EtherCAT)/Term 7 (EK1101)/Term 14 (EK1122)/Term 32 (EK1101)/NTTA1 - NTTA2 (N9) (EL7342)
//     Drive/Inputs/In/nState1 @bit 3 <-> DCM Status Channel 2/Status/Error
//     Drive/Inputs/In/nState1 @bit 5 <-> DCM Status Channel 2/Status/Moving negative
//     Drive/Inputs/In/nState1 @bit 4 <-> DCM Status Channel 2/Status/Moving positive
//     Drive/Inputs/In/nState1 @bit 1 <-> DCM Status Channel 2/Status/Ready
//     Drive/Inputs/In/nState1 <-> DCM Status Channel 2/Status/Ready to enable
//     Drive/Inputs/In/nState1 @bit 6 <-> DCM Status Channel 2/Status/Torque reduced
//     Drive/Inputs/In/nState1 @bit 2 <-> DCM Status Channel 2/Status/Warning
//     Drive/Inputs/In/nState2 @bit 3 <-> DCM Status Channel 2/Status/Digital input 1
//     Drive/Inputs/In/nState2 @bit 4 <-> DCM Status Channel 2/Status/Digital input 2
//     Drive/Inputs/In/nState2 @bit 5 <-> DCM Status Channel 2/Status/Sync error
//     Drive/Inputs/In/nState2 @bit 7 <-> DCM Status Channel 2/Status/TxPDO Toggle
//     Drive/Inputs/In/nState4 @bit 1 <-> WcState/InputToggle
//     Drive/Inputs/In/nState4 <-> WcState/WcState
//     Drive/Outputs/Out/nCtrl1 <-> DCM Control Channel 2/Control/Enable
//     Drive/Outputs/Out/nCtrl1 @bit 2 <-> DCM Control Channel 2/Control/Reduce torque
//     Drive/Outputs/Out/nCtrl1 @bit 1 <-> DCM Control Channel 2/Control/Reset
//     Drive/Outputs/Out/nCtrl1 @bit 3 <-> DCM Control Channel 2/Control/Threshold active
//     Drive/Outputs/Out/nDataOut2[0] <-> DCM Velocity Channel 2/Velocity
//     Enc/Inputs/In/nDataIn1[0] <-> ENC Status compact Channel 2/Counter value
//     Enc/Inputs/In/nDataIn2[0] <-> ENC Status compact Channel 2/Latch value
//     Enc/Inputs/In/nState1 @bit 4 <-> ENC Status compact Channel 2/Status/Counter overflow
//     Enc/Inputs/In/nState1 @bit 3 <-> ENC Status compact Channel 2/Status/Counter underflow
//     Enc/Inputs/In/nState1 @bit 7 <-> ENC Status compact Channel 2/Status/Extrapolation stall
//     Enc/Inputs/In/nState1 @bit 1 <-> ENC Status compact Channel 2/Status/Latch extern valid
//     Enc/Inputs/In/nState1 @bit 2 <-> ENC Status compact Channel 2/Status/Set counter done
//     Enc/Inputs/In/nState2 @bit 4 <-> ENC Status compact Channel 2/Status/Status of extern latch
//     Enc/Inputs/In/nState2 <-> ENC Status compact Channel 2/Status/Status of input A
//     Enc/Inputs/In/nState2 @bit 1 <-> ENC Status compact Channel 2/Status/Status of input B
//     Enc/Inputs/In/nState2 @bit 5 <-> ENC Status compact Channel 2/Status/Sync error
//     Enc/Inputs/In/nState2 @bit 7 <-> ENC Status compact Channel 2/Status/TxPDO Toggle
//     Enc/Inputs/In/nState4 @bit 1 <-> WcState/InputToggle
//     Enc/Inputs/In/nState4 <-> WcState/WcState
//     Enc/Outputs/Out/nCtrl1 @bit 3 <-> ENC Control compact Channel 2/Control/Enable latch extern on negative edge
//     Enc/Outputs/Out/nCtrl1 @bit 1 <-> ENC Control compact Channel 2/Control/Enable latch extern on positive edge
//     Enc/Outputs/Out/nCtrl1 @bit 2 <-> ENC Control compact Channel 2/Control/Set counter
//     Enc/Outputs/Out/nDataOut1[0] <-> ENC Control compact Channel 2/Set counter value
//   NC-Task 1 SAF/Axes/NTTA3 <-> Device 1 (EtherCAT)/Term 7 (EK1101)/Term 14 (EK1122)/Term 32 (EK1101)/NTTA3 - NTTA4 (N10) (EL7342)
//     Drive/Inputs/In/nState1 @bit 3 <-> DCM Status Channel 1/Status/Error
//     Drive/Inputs/In/nState1 @bit 5 <-> DCM Status Channel 1/Status/Moving negative
//     Drive/Inputs/In/nState1 @bit 4 <-> DCM Status Channel 1/Status/Moving positive
//     Drive/Inputs/In/nState1 @bit 1 <-> DCM Status Channel 1/Status/Ready
//     Drive/Inputs/In/nState1 <-> DCM Status Channel 1/Status/Ready to enable
//     Drive/Inputs/In/nState1 @bit 6 <-> DCM Status Channel 1/Status/Torque reduced
//     Drive/Inputs/In/nState1 @bit 2 <-> DCM Status Channel 1/Status/Warning
//     Drive/Inputs/In/nState2 @bit 3 <-> DCM Status Channel 1/Status/Digital input 1
//     Drive/Inputs/In/nState2 @bit 4 <-> DCM Status Channel 1/Status/Digital input 2
//     Drive/Inputs/In/nState2 @bit 5 <-> DCM Status Channel 1/Status/Sync error
//     Drive/Inputs/In/nState2 @bit 7 <-> DCM Status Channel 1/Status/TxPDO Toggle
//     Drive/Inputs/In/nState4 @bit 1 <-> WcState/InputToggle
//     Drive/Inputs/In/nState4 <-> WcState/WcState
//     Drive/Outputs/Out/nCtrl1 <-> DCM Control Channel 1/Control/Enable
//     Drive/Outputs/Out/nCtrl1 @bit 2 <-> DCM Control Channel 1/Control/Reduce torque
//     Drive/Outputs/Out/nCtrl1 @bit 1 <-> DCM Control Channel 1/Control/Reset
//     Drive/Outputs/Out/nCtrl1 @bit 3 <-> DCM Control Channel 1/Control/Threshold active
//     Drive/Outputs/Out/nDataOut2[0] <-> DCM Velocity Channel 1/Velocity
//     Enc/Inputs/In/nDataIn1[0] <-> ENC Status compact Channel 1/Counter value
//     Enc/Inputs/In/nDataIn2[0] <-> ENC Status compact Channel 1/Latch value
//     Enc/Inputs/In/nState1 @bit 4 <-> ENC Status compact Channel 1/Status/Counter overflow
//     Enc/Inputs/In/nState1 @bit 3 <-> ENC Status compact Channel 1/Status/Counter underflow
//     Enc/Inputs/In/nState1 @bit 7 <-> ENC Status compact Channel 1/Status/Extrapolation stall
//     Enc/Inputs/In/nState1 @bit 1 <-> ENC Status compact Channel 1/Status/Latch extern valid
//     Enc/Inputs/In/nState1 @bit 2 <-> ENC Status compact Channel 1/Status/Set counter done
//     Enc/Inputs/In/nState2 @bit 4 <-> ENC Status compact Channel 1/Status/Status of extern latch
//     Enc/Inputs/In/nState2 <-> ENC Status compact Channel 1/Status/Status of input A
//     Enc/Inputs/In/nState2 @bit 1 <-> ENC Status compact Channel 1/Status/Status of input B
//     Enc/Inputs/In/nState2 @bit 5 <-> ENC Status compact Channel 1/Status/Sync error
//     Enc/Inputs/In/nState2 @bit 7 <-> ENC Status compact Channel 1/Status/TxPDO Toggle
//     Enc/Inputs/In/nState4 @bit 1 <-> WcState/InputToggle
//     Enc/Inputs/In/nState4 <-> WcState/WcState
//     Enc/Outputs/Out/nCtrl1 @bit 3 <-> ENC Control compact Channel 1/Control/Enable latch extern on negative edge
//     Enc/Outputs/Out/nCtrl1 @bit 1 <-> ENC Control compact Channel 1/Control/Enable latch extern on positive edge
//     Enc/Outputs/Out/nCtrl1 @bit 2 <-> ENC Control compact Channel 1/Control/Set counter
//     Enc/Outputs/Out/nDataOut1[0] <-> ENC Control compact Channel 1/Set counter value
//   NC-Task 1 SAF/Axes/NTTA4 <-> Device 1 (EtherCAT)/Term 7 (EK1101)/Term 14 (EK1122)/Term 32 (EK1101)/NTTA3 - NTTA4 (N10) (EL7342)
//     Drive/Inputs/In/nState1 @bit 3 <-> DCM Status Channel 2/Status/Error
//     Drive/Inputs/In/nState1 @bit 5 <-> DCM Status Channel 2/Status/Moving negative
//     Drive/Inputs/In/nState1 @bit 4 <-> DCM Status Channel 2/Status/Moving positive
//     Drive/Inputs/In/nState1 @bit 1 <-> DCM Status Channel 2/Status/Ready
//     Drive/Inputs/In/nState1 <-> DCM Status Channel 2/Status/Ready to enable
//     Drive/Inputs/In/nState1 @bit 6 <-> DCM Status Channel 2/Status/Torque reduced
//     Drive/Inputs/In/nState1 @bit 2 <-> DCM Status Channel 2/Status/Warning
//     Drive/Inputs/In/nState2 @bit 3 <-> DCM Status Channel 2/Status/Digital input 1
//     Drive/Inputs/In/nState2 @bit 4 <-> DCM Status Channel 2/Status/Digital input 2
//     Drive/Inputs/In/nState2 @bit 5 <-> DCM Status Channel 2/Status/Sync error
//     Drive/Inputs/In/nState2 @bit 7 <-> DCM Status Channel 2/Status/TxPDO Toggle
//     Drive/Inputs/In/nState4 @bit 1 <-> WcState/InputToggle
//     Drive/Inputs/In/nState4 <-> WcState/WcState
//     Drive/Outputs/Out/nCtrl1 <-> DCM Control Channel 2/Control/Enable
//     Drive/Outputs/Out/nCtrl1 @bit 2 <-> DCM Control Channel 2/Control/Reduce torque
//     Drive/Outputs/Out/nCtrl1 @bit 1 <-> DCM Control Channel 2/Control/Reset
//     Drive/Outputs/Out/nCtrl1 @bit 3 <-> DCM Control Channel 2/Control/Threshold active
//     Drive/Outputs/Out/nDataOut2[0] <-> DCM Velocity Channel 2/Velocity
//     Enc/Inputs/In/nDataIn1[0] <-> ENC Status compact Channel 2/Counter value
//     Enc/Inputs/In/nDataIn2[0] <-> ENC Status compact Channel 2/Latch value
//     Enc/Inputs/In/nState1 @bit 4 <-> ENC Status compact Channel 2/Status/Counter overflow
//     Enc/Inputs/In/nState1 @bit 3 <-> ENC Status compact Channel 2/Status/Counter underflow
//     Enc/Inputs/In/nState1 @bit 7 <-> ENC Status compact Channel 2/Status/Extrapolation stall
//     Enc/Inputs/In/nState1 @bit 1 <-> ENC Status compact Channel 2/Status/Latch extern valid
//     Enc/Inputs/In/nState1 @bit 2 <-> ENC Status compact Channel 2/Status/Set counter done
//     Enc/Inputs/In/nState2 @bit 4 <-> ENC Status compact Channel 2/Status/Status of extern latch
//     Enc/Inputs/In/nState2 <-> ENC Status compact Channel 2/Status/Status of input A
//     Enc/Inputs/In/nState2 @bit 1 <-> ENC Status compact Channel 2/Status/Status of input B
//     Enc/Inputs/In/nState2 @bit 5 <-> ENC Status compact Channel 2/Status/Sync error
//     Enc/Inputs/In/nState2 @bit 7 <-> ENC Status compact Channel 2/Status/TxPDO Toggle
//     Enc/Inputs/In/nState4 @bit 1 <-> WcState/InputToggle
//     Enc/Inputs/In/nState4 <-> WcState/WcState
//     Enc/Outputs/Out/nCtrl1 @bit 3 <-> ENC Control compact Channel 2/Control/Enable latch extern on negative edge
//     Enc/Outputs/Out/nCtrl1 @bit 1 <-> ENC Control compact Channel 2/Control/Enable latch extern on positive edge
//     Enc/Outputs/Out/nCtrl1 @bit 2 <-> ENC Control compact Channel 2/Control/Set counter
//     Enc/Outputs/Out/nDataOut1[0] <-> ENC Control compact Channel 2/Set counter value
//   NC-Task 1 SAF/Axes/NTTB1 <-> Device 1 (EtherCAT)/Term 7 (EK1101)/Term 14 (EK1122)/Term 32 (EK1101)/NTTB1 - NTTB2 (N18) (EL7342)
//     Drive/Inputs/In/nState1 @bit 3 <-> DCM Status Channel 1/Status/Error
//     Drive/Inputs/In/nState1 @bit 5 <-> DCM Status Channel 1/Status/Moving negative
//     Drive/Inputs/In/nState1 @bit 4 <-> DCM Status Channel 1/Status/Moving positive
//     Drive/Inputs/In/nState1 @bit 1 <-> DCM Status Channel 1/Status/Ready
//     Drive/Inputs/In/nState1 <-> DCM Status Channel 1/Status/Ready to enable
//     Drive/Inputs/In/nState1 @bit 6 <-> DCM Status Channel 1/Status/Torque reduced
//     Drive/Inputs/In/nState1 @bit 2 <-> DCM Status Channel 1/Status/Warning
//     Drive/Inputs/In/nState2 @bit 3 <-> DCM Status Channel 1/Status/Digital input 1
//     Drive/Inputs/In/nState2 @bit 4 <-> DCM Status Channel 1/Status/Digital input 2
//     Drive/Inputs/In/nState2 @bit 5 <-> DCM Status Channel 1/Status/Sync error
//     Drive/Inputs/In/nState2 @bit 7 <-> DCM Status Channel 1/Status/TxPDO Toggle
//     Drive/Inputs/In/nState4 @bit 1 <-> WcState/InputToggle
//     Drive/Inputs/In/nState4 <-> WcState/WcState
//     Drive/Outputs/Out/nCtrl1 <-> DCM Control Channel 1/Control/Enable
//     Drive/Outputs/Out/nCtrl1 @bit 2 <-> DCM Control Channel 1/Control/Reduce torque
//     Drive/Outputs/Out/nCtrl1 @bit 1 <-> DCM Control Channel 1/Control/Reset
//     Drive/Outputs/Out/nCtrl1 @bit 3 <-> DCM Control Channel 1/Control/Threshold active
//     Drive/Outputs/Out/nDataOut2[0] <-> DCM Velocity Channel 1/Velocity
//     Enc/Inputs/In/nDataIn1[0] <-> ENC Status compact Channel 1/Counter value
//     Enc/Inputs/In/nDataIn2[0] <-> ENC Status compact Channel 1/Latch value
//     Enc/Inputs/In/nState1 @bit 4 <-> ENC Status compact Channel 1/Status/Counter overflow
//     Enc/Inputs/In/nState1 @bit 3 <-> ENC Status compact Channel 1/Status/Counter underflow
//     Enc/Inputs/In/nState1 @bit 7 <-> ENC Status compact Channel 1/Status/Extrapolation stall
//     Enc/Inputs/In/nState1 @bit 1 <-> ENC Status compact Channel 1/Status/Latch extern valid
//     Enc/Inputs/In/nState1 @bit 2 <-> ENC Status compact Channel 1/Status/Set counter done
//     Enc/Inputs/In/nState2 @bit 4 <-> ENC Status compact Channel 1/Status/Status of extern latch
//     Enc/Inputs/In/nState2 <-> ENC Status compact Channel 1/Status/Status of input A
//     Enc/Inputs/In/nState2 @bit 1 <-> ENC Status compact Channel 1/Status/Status of input B
//     Enc/Inputs/In/nState2 @bit 5 <-> ENC Status compact Channel 1/Status/Sync error
//     Enc/Inputs/In/nState2 @bit 7 <-> ENC Status compact Channel 1/Status/TxPDO Toggle
//     Enc/Inputs/In/nState4 @bit 1 <-> WcState/InputToggle
//     Enc/Inputs/In/nState4 <-> WcState/WcState
//     Enc/Outputs/Out/nCtrl1 @bit 3 <-> ENC Control compact Channel 1/Control/Enable latch extern on negative edge
//     Enc/Outputs/Out/nCtrl1 @bit 1 <-> ENC Control compact Channel 1/Control/Enable latch extern on positive edge
//     Enc/Outputs/Out/nCtrl1 @bit 2 <-> ENC Control compact Channel 1/Control/Set counter
//     Enc/Outputs/Out/nDataOut1[0] <-> ENC Control compact Channel 1/Set counter value
//   NC-Task 1 SAF/Axes/NTTB2 <-> Device 1 (EtherCAT)/Term 7 (EK1101)/Term 14 (EK1122)/Term 32 (EK1101)/NTTB1 - NTTB2 (N18) (EL7342)
//     Drive/Inputs/In/nState1 @bit 3 <-> DCM Status Channel 2/Status/Error
//     Drive/Inputs/In/nState1 @bit 5 <-> DCM Status Channel 2/Status/Moving negative
//     Drive/Inputs/In/nState1 @bit 4 <-> DCM Status Channel 2/Status/Moving positive
//     Drive/Inputs/In/nState1 @bit 1 <-> DCM Status Channel 2/Status/Ready
//     Drive/Inputs/In/nState1 <-> DCM Status Channel 2/Status/Ready to enable
//     Drive/Inputs/In/nState1 @bit 6 <-> DCM Status Channel 2/Status/Torque reduced
//     Drive/Inputs/In/nState1 @bit 2 <-> DCM Status Channel 2/Status/Warning
//     Drive/Inputs/In/nState2 @bit 3 <-> DCM Status Channel 2/Status/Digital input 1
//     Drive/Inputs/In/nState2 @bit 4 <-> DCM Status Channel 2/Status/Digital input 2
//     Drive/Inputs/In/nState2 @bit 5 <-> DCM Status Channel 2/Status/Sync error
//     Drive/Inputs/In/nState2 @bit 7 <-> DCM Status Channel 2/Status/TxPDO Toggle
//     Drive/Inputs/In/nState4 @bit 1 <-> WcState/InputToggle
//     Drive/Inputs/In/nState4 <-> WcState/WcState
//     Drive/Outputs/Out/nCtrl1 <-> DCM Control Channel 2/Control/Enable
//     Drive/Outputs/Out/nCtrl1 @bit 2 <-> DCM Control Channel 2/Control/Reduce torque
//     Drive/Outputs/Out/nCtrl1 @bit 1 <-> DCM Control Channel 2/Control/Reset
//     Drive/Outputs/Out/nCtrl1 @bit 3 <-> DCM Control Channel 2/Control/Threshold active
//     Drive/Outputs/Out/nDataOut2[0] <-> DCM Velocity Channel 2/Velocity
//     Enc/Inputs/In/nDataIn1[0] <-> ENC Status compact Channel 2/Counter value
//     Enc/Inputs/In/nDataIn2[0] <-> ENC Status compact Channel 2/Latch value
//     Enc/Inputs/In/nState1 @bit 4 <-> ENC Status compact Channel 2/Status/Counter overflow
//     Enc/Inputs/In/nState1 @bit 3 <-> ENC Status compact Channel 2/Status/Counter underflow
//     Enc/Inputs/In/nState1 @bit 7 <-> ENC Status compact Channel 2/Status/Extrapolation stall
//     Enc/Inputs/In/nState1 @bit 1 <-> ENC Status compact Channel 2/Status/Latch extern valid
//     Enc/Inputs/In/nState1 @bit 2 <-> ENC Status compact Channel 2/Status/Set counter done
//     Enc/Inputs/In/nState2 @bit 4 <-> ENC Status compact Channel 2/Status/Status of extern latch
//     Enc/Inputs/In/nState2 <-> ENC Status compact Channel 2/Status/Status of input A
//     Enc/Inputs/In/nState2 @bit 1 <-> ENC Status compact Channel 2/Status/Status of input B
//     Enc/Inputs/In/nState2 @bit 5 <-> ENC Status compact Channel 2/Status/Sync error
//     Enc/Inputs/In/nState2 @bit 7 <-> ENC Status compact Channel 2/Status/TxPDO Toggle
//     Enc/Inputs/In/nState4 @bit 1 <-> WcState/InputToggle
//     Enc/Inputs/In/nState4 <-> WcState/WcState
//     Enc/Outputs/Out/nCtrl1 @bit 3 <-> ENC Control compact Channel 2/Control/Enable latch extern on negative edge
//     Enc/Outputs/Out/nCtrl1 @bit 1 <-> ENC Control compact Channel 2/Control/Enable latch extern on positive edge
//     Enc/Outputs/Out/nCtrl1 @bit 2 <-> ENC Control compact Channel 2/Control/Set counter
//     Enc/Outputs/Out/nDataOut1[0] <-> ENC Control compact Channel 2/Set counter value
//   NC-Task 1 SAF/Axes/NTTB3 <-> Device 1 (EtherCAT)/Term 7 (EK1101)/Term 14 (EK1122)/Term 32 (EK1101)/NTTB3 - NTTB4 (N19) (EL7342)
//     Drive/Inputs/In/nState1 @bit 3 <-> DCM Status Channel 1/Status/Error
//     Drive/Inputs/In/nState1 @bit 5 <-> DCM Status Channel 1/Status/Moving negative
//     Drive/Inputs/In/nState1 @bit 4 <-> DCM Status Channel 1/Status/Moving positive
//     Drive/Inputs/In/nState1 @bit 1 <-> DCM Status Channel 1/Status/Ready
//     Drive/Inputs/In/nState1 <-> DCM Status Channel 1/Status/Ready to enable
//     Drive/Inputs/In/nState1 @bit 6 <-> DCM Status Channel 1/Status/Torque reduced
//     Drive/Inputs/In/nState1 @bit 2 <-> DCM Status Channel 1/Status/Warning
//     Drive/Inputs/In/nState2 @bit 3 <-> DCM Status Channel 1/Status/Digital input 1
//     Drive/Inputs/In/nState2 @bit 4 <-> DCM Status Channel 1/Status/Digital input 2
//     Drive/Inputs/In/nState2 @bit 5 <-> DCM Status Channel 1/Status/Sync error
//     Drive/Inputs/In/nState2 @bit 7 <-> DCM Status Channel 1/Status/TxPDO Toggle
//     Drive/Inputs/In/nState4 @bit 1 <-> WcState/InputToggle
//     Drive/Inputs/In/nState4 <-> WcState/WcState
//     Drive/Outputs/Out/nCtrl1 <-> DCM Control Channel 1/Control/Enable
//     Drive/Outputs/Out/nCtrl1 @bit 2 <-> DCM Control Channel 1/Control/Reduce torque
//     Drive/Outputs/Out/nCtrl1 @bit 1 <-> DCM Control Channel 1/Control/Reset
//     Drive/Outputs/Out/nCtrl1 @bit 3 <-> DCM Control Channel 1/Control/Threshold active
//     Drive/Outputs/Out/nDataOut2[0] <-> DCM Velocity Channel 1/Velocity
//     Enc/Inputs/In/nDataIn1[0] <-> ENC Status compact Channel 1/Counter value
//     Enc/Inputs/In/nDataIn2[0] <-> ENC Status compact Channel 1/Latch value
//     Enc/Inputs/In/nState1 @bit 4 <-> ENC Status compact Channel 1/Status/Counter overflow
//     Enc/Inputs/In/nState1 @bit 3 <-> ENC Status compact Channel 1/Status/Counter underflow
//     Enc/Inputs/In/nState1 @bit 7 <-> ENC Status compact Channel 1/Status/Extrapolation stall
//     Enc/Inputs/In/nState1 @bit 1 <-> ENC Status compact Channel 1/Status/Latch extern valid
//     Enc/Inputs/In/nState1 @bit 2 <-> ENC Status compact Channel 1/Status/Set counter done
//     Enc/Inputs/In/nState2 @bit 4 <-> ENC Status compact Channel 1/Status/Status of extern latch
//     Enc/Inputs/In/nState2 <-> ENC Status compact Channel 1/Status/Status of input A
//     Enc/Inputs/In/nState2 @bit 1 <-> ENC Status compact Channel 1/Status/Status of input B
//     Enc/Inputs/In/nState2 @bit 5 <-> ENC Status compact Channel 1/Status/Sync error
//     Enc/Inputs/In/nState2 @bit 7 <-> ENC Status compact Channel 1/Status/TxPDO Toggle
//     Enc/Inputs/In/nState4 @bit 1 <-> WcState/InputToggle
//     Enc/Inputs/In/nState4 <-> WcState/WcState
//     Enc/Outputs/Out/nCtrl1 @bit 3 <-> ENC Control compact Channel 1/Control/Enable latch extern on negative edge
//     Enc/Outputs/Out/nCtrl1 @bit 1 <-> ENC Control compact Channel 1/Control/Enable latch extern on positive edge
//     Enc/Outputs/Out/nCtrl1 @bit 2 <-> ENC Control compact Channel 1/Control/Set counter
//     Enc/Outputs/Out/nDataOut1[0] <-> ENC Control compact Channel 1/Set counter value
//   NC-Task 1 SAF/Axes/NTTB4 <-> Device 1 (EtherCAT)/Term 7 (EK1101)/Term 14 (EK1122)/Term 32 (EK1101)/NTTB3 - NTTB4 (N19) (EL7342)
//     Drive/Inputs/In/nState1 @bit 3 <-> DCM Status Channel 2/Status/Error
//     Drive/Inputs/In/nState1 @bit 5 <-> DCM Status Channel 2/Status/Moving negative
//     Drive/Inputs/In/nState1 @bit 4 <-> DCM Status Channel 2/Status/Moving positive
//     Drive/Inputs/In/nState1 @bit 1 <-> DCM Status Channel 2/Status/Ready
//     Drive/Inputs/In/nState1 <-> DCM Status Channel 2/Status/Ready to enable
//     Drive/Inputs/In/nState1 @bit 6 <-> DCM Status Channel 2/Status/Torque reduced
//     Drive/Inputs/In/nState1 @bit 2 <-> DCM Status Channel 2/Status/Warning
//     Drive/Inputs/In/nState2 @bit 3 <-> DCM Status Channel 2/Status/Digital input 1
//     Drive/Inputs/In/nState2 @bit 4 <-> DCM Status Channel 2/Status/Digital input 2
//     Drive/Inputs/In/nState2 @bit 5 <-> DCM Status Channel 2/Status/Sync error
//     Drive/Inputs/In/nState2 @bit 7 <-> DCM Status Channel 2/Status/TxPDO Toggle
//     Drive/Inputs/In/nState4 @bit 1 <-> WcState/InputToggle
//     Drive/Inputs/In/nState4 <-> WcState/WcState
//     Drive/Outputs/Out/nCtrl1 <-> DCM Control Channel 2/Control/Enable
//     Drive/Outputs/Out/nCtrl1 @bit 2 <-> DCM Control Channel 2/Control/Reduce torque
//     Drive/Outputs/Out/nCtrl1 @bit 1 <-> DCM Control Channel 2/Control/Reset
//     Drive/Outputs/Out/nCtrl1 @bit 3 <-> DCM Control Channel 2/Control/Threshold active
//     Drive/Outputs/Out/nDataOut2[0] <-> DCM Velocity Channel 2/Velocity
//     Enc/Inputs/In/nDataIn1[0] <-> ENC Status compact Channel 2/Counter value
//     Enc/Inputs/In/nDataIn2[0] <-> ENC Status compact Channel 2/Latch value
//     Enc/Inputs/In/nState1 @bit 4 <-> ENC Status compact Channel 2/Status/Counter overflow
//     Enc/Inputs/In/nState1 @bit 3 <-> ENC Status compact Channel 2/Status/Counter underflow
//     Enc/Inputs/In/nState1 @bit 7 <-> ENC Status compact Channel 2/Status/Extrapolation stall
//     Enc/Inputs/In/nState1 @bit 1 <-> ENC Status compact Channel 2/Status/Latch extern valid
//     Enc/Inputs/In/nState1 @bit 2 <-> ENC Status compact Channel 2/Status/Set counter done
//     Enc/Inputs/In/nState2 @bit 4 <-> ENC Status compact Channel 2/Status/Status of extern latch
//     Enc/Inputs/In/nState2 <-> ENC Status compact Channel 2/Status/Status of input A
//     Enc/Inputs/In/nState2 @bit 1 <-> ENC Status compact Channel 2/Status/Status of input B
//     Enc/Inputs/In/nState2 @bit 5 <-> ENC Status compact Channel 2/Status/Sync error
//     Enc/Inputs/In/nState2 @bit 7 <-> ENC Status compact Channel 2/Status/TxPDO Toggle
//     Enc/Inputs/In/nState4 @bit 1 <-> WcState/InputToggle
//     Enc/Inputs/In/nState4 <-> WcState/WcState
//     Enc/Outputs/Out/nCtrl1 @bit 3 <-> ENC Control compact Channel 2/Control/Enable latch extern on negative edge
//     Enc/Outputs/Out/nCtrl1 @bit 1 <-> ENC Control compact Channel 2/Control/Enable latch extern on positive edge
//     Enc/Outputs/Out/nCtrl1 @bit 2 <-> ENC Control compact Channel 2/Control/Set counter
//     Enc/Outputs/Out/nDataOut1[0] <-> ENC Control compact Channel 2/Set counter value
//   nott_ics/nott_ics Instance <-> Device 1 (EtherCAT)
//     PlcTask Inputs/MAIN.fbServices.i_nDevState <-> Inputs/DevState
//   nott_ics/nott_ics Instance <-> Device 1 (EtherCAT)/Term 1 (EK1200)/Term 4 (EL2008)
//     PlcTask Outputs/MAIN.nott_ics.CO2_Pressure_Control.CO2_Valve.Actuator.q_bCtrl <-> Channel 1/Output
//   nott_ics/nott_ics Instance <-> Device 1 (EtherCAT)/Term 7 (EK1101)/Term 14 (EK1122)/Term 15 (EK1101)/N13 (EL1008)
//     PlcTask Inputs/MAIN.nott_ics.Birefringence.NPC1.switches/bREF <-> Channel 1/Input
//     PlcTask Inputs/MAIN.nott_ics.Birefringence.NPC2.switches/bLHW <-> Channel 3/Input
//     PlcTask Inputs/MAIN.nott_ics.Birefringence.NPC3.switches/bLHW <-> Channel 5/Input
//     PlcTask Inputs/MAIN.nott_ics.Birefringence.NPC4.switches/bLHW <-> Channel 7/Input
//     PlcTask Inputs/MAIN.nott_ics.Birefringence.NPC2.switches/bUHW <-> Channel 4/Input
//     PlcTask Inputs/MAIN.nott_ics.Birefringence.NPC3.switches/bUHW <-> Channel 6/Input
//     PlcTask Inputs/MAIN.nott_ics.Birefringence.NPC4.switches/bUHW <-> Channel 8/Input
//   nott_ics/nott_ics Instance <-> Device 1 (EtherCAT)/Term 7 (EK1101)/Term 14 (EK1122)/Term 15 (EK1101)/N3 (EL1008)
//     PlcTask Inputs/MAIN.nott_ics.CO2TransStages.NCP{1..4}.switches/bLHW <-> Channel {1..7 step 2}/Input  (4 links)
//     PlcTask Inputs/MAIN.nott_ics.CO2TransStages.NCP{1..4}.switches/bUHW <-> Channel {2..8 step 2}/Input  (4 links)
//   nott_ics/nott_ics Instance <-> Device 1 (EtherCAT)/Term 7 (EK1101)/Term 14 (EK1122)/Term 15 (EK1101)/N7 (EL1008)
//     PlcTask Inputs/MAIN.nott_ics.ZnSeActuators.NGP{1..4}.switches/bLHW <-> Channel {1..7 step 2}/Input  (4 links)
//     PlcTask Inputs/MAIN.nott_ics.ZnSeActuators.NGP{1..4}.switches/bUHW <-> Channel {2..8 step 2}/Input  (4 links)
//   nott_ics/nott_ics Instance <-> Device 1 (EtherCAT)/Term 7 (EK1101)/Term 14 (EK1122)/Term 15 (EK1101)/N9 (EL1008)
//     PlcTask Inputs/MAIN.nott_ics.Calibration_Unit_Beam_Splitter.NBS.switches/bLHW <-> Channel 1/Input
//     PlcTask Inputs/MAIN.nott_ics.Calibration_Unit_Beam_Splitter.NBS.switches/bUHW <-> Channel 2/Input
//   nott_ics/nott_ics Instance <-> Device 1 (EtherCAT)/Term 7 (EK1101)/Term 14 (EK1122)/Term 15 (EK1101)/NBS (N8) (EL7342)
//     PlcTask Inputs/MAIN.nott_ics.Calibration_Unit_Beam_Splitter.NBS.i_nCouplerState <-> InfoData/State
//   nott_ics/nott_ics Instance <-> Device 1 (EtherCAT)/Term 7 (EK1101)/Term 14 (EK1122)/Term 15 (EK1101)/NCP1 - NCP2 (N1) (EL7342)
//     PlcTask Inputs/MAIN.nott_ics.CO2TransStages.NCP1.i_nCouplerState <-> InfoData/State
//     PlcTask Inputs/MAIN.nott_ics.CO2TransStages.NCP2.i_nCouplerState <-> InfoData/State
//   nott_ics/nott_ics Instance <-> Device 1 (EtherCAT)/Term 7 (EK1101)/Term 14 (EK1122)/Term 15 (EK1101)/NCP3 - NCP4 (N2) (EL7342)
//     PlcTask Inputs/MAIN.nott_ics.CO2TransStages.NCP3.i_nCouplerState <-> InfoData/State
//     PlcTask Inputs/MAIN.nott_ics.CO2TransStages.NCP4.i_nCouplerState <-> InfoData/State
//   nott_ics/nott_ics Instance <-> Device 1 (EtherCAT)/Term 7 (EK1101)/Term 14 (EK1122)/Term 15 (EK1101)/NGP1 - NGP2 (N5) (EL7342)
//     PlcTask Inputs/MAIN.nott_ics.ZnSeActuators.NGP1.i_nCouplerState <-> InfoData/State
//     PlcTask Inputs/MAIN.nott_ics.ZnSeActuators.NGP2.i_nCouplerState <-> InfoData/State
//   nott_ics/nott_ics Instance <-> Device 1 (EtherCAT)/Term 7 (EK1101)/Term 14 (EK1122)/Term 15 (EK1101)/NGP3 - NGP4 (N6) (EL7342)
//     PlcTask Inputs/MAIN.nott_ics.ZnSeActuators.NGP3.i_nCouplerState <-> InfoData/State
//     PlcTask Inputs/MAIN.nott_ics.ZnSeActuators.NGP4.i_nCouplerState <-> InfoData/State
//   nott_ics/nott_ics Instance <-> Device 1 (EtherCAT)/Term 7 (EK1101)/Term 14 (EK1122)/Term 15 (EK1101)/NPC1 - NPC2 (N11) (EL7342)
//     PlcTask Inputs/MAIN.nott_ics.Birefringence.NPC1.i_nCouplerState <-> InfoData/State
//     PlcTask Inputs/MAIN.nott_ics.Birefringence.NPC2.i_nCouplerState <-> InfoData/State
//   nott_ics/nott_ics Instance <-> Device 1 (EtherCAT)/Term 7 (EK1101)/Term 14 (EK1122)/Term 15 (EK1101)/NPC3 - NPC4 (N12) (EL7342)
//     PlcTask Inputs/MAIN.nott_ics.Birefringence.NPC3.i_nCouplerState <-> InfoData/State
//     PlcTask Inputs/MAIN.nott_ics.Birefringence.NPC4.i_nCouplerState <-> InfoData/State
//   nott_ics/nott_ics Instance <-> Device 1 (EtherCAT)/Term 7 (EK1101)/Term 14 (EK1122)/Term 15 (EK1101)/NSH1 (N16) (EL7047)
//     PlcTask Inputs/MAIN.nott_ics.Shutters.NSH1.i_nCouplerState <-> InfoData/State
//     PlcTask Inputs/MAIN.nott_ics.Shutters.NSH1.switches/bLHW <-> STM Status/Status/Digital input 1
//     PlcTask Inputs/MAIN.nott_ics.Shutters.NSH1.switches/bUHW <-> STM Status/Status/Digital input 2
//     PlcTask Inputs/MAIN.nott_ics.Shutters.Test_Shutter.i_nCouplerState <-> InfoData/State
//   nott_ics/nott_ics Instance <-> Device 1 (EtherCAT)/Term 7 (EK1101)/Term 14 (EK1122)/Term 15 (EK1101)/NSH2 (N17) (EL7047)
//     PlcTask Inputs/MAIN.nott_ics.Shutters.NSH2.i_nCouplerState <-> InfoData/State
//     PlcTask Inputs/MAIN.nott_ics.Shutters.NSH2.switches/bLHW <-> STM Status/Status/Digital input 1
//     PlcTask Inputs/MAIN.nott_ics.Shutters.NSH2.switches/bUHW <-> STM Status/Status/Digital input 2
//   nott_ics/nott_ics Instance <-> Device 1 (EtherCAT)/Term 7 (EK1101)/Term 14 (EK1122)/Term 15 (EK1101)/NSH3 (N18) (EL7047)
//     PlcTask Inputs/MAIN.nott_ics.Shutters.NSH3.i_nCouplerState <-> InfoData/State
//     PlcTask Inputs/MAIN.nott_ics.Shutters.NSH3.switches/bLHW <-> STM Status/Status/Digital input 1
//     PlcTask Inputs/MAIN.nott_ics.Shutters.NSH3.switches/bUHW <-> STM Status/Status/Digital input 2
//   nott_ics/nott_ics Instance <-> Device 1 (EtherCAT)/Term 7 (EK1101)/Term 14 (EK1122)/Term 15 (EK1101)/NSH4 (N19) (EL7047)
//     PlcTask Inputs/MAIN.nott_ics.Shutters.NSH4.i_nCouplerState <-> InfoData/State
//     PlcTask Inputs/MAIN.nott_ics.Shutters.NSH4.switches/bLHW <-> STM Status/Status/Digital input 1
//     PlcTask Inputs/MAIN.nott_ics.Shutters.NSH4.switches/bUHW <-> STM Status/Status/Digital input 2
//   nott_ics/nott_ics Instance <-> Device 1 (EtherCAT)/Term 7 (EK1101)/Term 14 (EK1122)/Term 32 (EK1101)/N11 (EL1008)
//     PlcTask Inputs/MAIN.nott_ics.TipTilt.NTTA{1..4}.switches/bLHW <-> Channel {1..7 step 2}/Input  (4 links)
//     PlcTask Inputs/MAIN.nott_ics.TipTilt.NTTA{1..4}.switches/bUHW <-> Channel {2..8 step 2}/Input  (4 links)
//   nott_ics/nott_ics Instance <-> Device 1 (EtherCAT)/Term 7 (EK1101)/Term 14 (EK1122)/Term 32 (EK1101)/N16 (EL1008)
//     PlcTask Inputs/MAIN.nott_ics.TipTilt.NTPB{1..4}.switches/bLHW <-> Channel {1..7 step 2}/Input  (4 links)
//     PlcTask Inputs/MAIN.nott_ics.TipTilt.NTPB{1..4}.switches/bUHW <-> Channel {2..8 step 2}/Input  (4 links)
//   nott_ics/nott_ics Instance <-> Device 1 (EtherCAT)/Term 7 (EK1101)/Term 14 (EK1122)/Term 32 (EK1101)/N20 (EL1008)
//     PlcTask Inputs/MAIN.nott_ics.TipTilt.NTTB{1..4}.switches/bLHW <-> Channel {1..7 step 2}/Input  (4 links)
//     PlcTask Inputs/MAIN.nott_ics.TipTilt.NTTB{1..4}.switches/bUHW <-> Channel {2..8 step 2}/Input  (4 links)
//   nott_ics/nott_ics Instance <-> Device 1 (EtherCAT)/Term 7 (EK1101)/Term 14 (EK1122)/Term 32 (EK1101)/N8 (EL1008)
//     PlcTask Inputs/MAIN.nott_ics.TipTilt.NTPA{1..4}.switches/bLHW <-> Channel {1..7 step 2}/Input  (4 links)
//     PlcTask Inputs/MAIN.nott_ics.TipTilt.NTPA{1..4}.switches/bUHW <-> Channel {2..8 step 2}/Input  (4 links)
//   nott_ics/nott_ics Instance <-> Device 1 (EtherCAT)/Term 7 (EK1101)/Term 14 (EK1122)/Term 32 (EK1101)/NDL1 (N1) (EL7047)
//     PlcTask Inputs/MAIN.nott_ics.Delay_Lines.NDL1.i_nCouplerState <-> InfoData/State
//     PlcTask Inputs/MAIN.nott_ics.Delay_Lines.NDL1.switches/bLHW <-> STM Status/Status/Digital input 1
//     PlcTask Inputs/MAIN.nott_ics.Delay_Lines.NDL1.switches/bUHW <-> STM Status/Status/Digital input 2
//   nott_ics/nott_ics Instance <-> Device 1 (EtherCAT)/Term 7 (EK1101)/Term 14 (EK1122)/Term 32 (EK1101)/NDL2 (N2) (EL7047)
//     PlcTask Inputs/MAIN.nott_ics.Delay_Lines.NDL2.i_nCouplerState <-> InfoData/State
//     PlcTask Inputs/MAIN.nott_ics.Delay_Lines.NDL2.switches/bLHW <-> STM Status/Status/Digital input 1
//     PlcTask Inputs/MAIN.nott_ics.Delay_Lines.NDL2.switches/bUHW <-> STM Status/Status/Digital input 2
//   nott_ics/nott_ics Instance <-> Device 1 (EtherCAT)/Term 7 (EK1101)/Term 14 (EK1122)/Term 32 (EK1101)/NDL3 (N3) (EL7047)
//     PlcTask Inputs/MAIN.nott_ics.Delay_Lines.NDL3.i_nCouplerState <-> InfoData/State
//     PlcTask Inputs/MAIN.nott_ics.Delay_Lines.NDL3.switches/bLHW <-> STM Status/Status/Digital input 1
//     PlcTask Inputs/MAIN.nott_ics.Delay_Lines.NDL3.switches/bUHW <-> STM Status/Status/Digital input 2
//   nott_ics/nott_ics Instance <-> Device 1 (EtherCAT)/Term 7 (EK1101)/Term 14 (EK1122)/Term 32 (EK1101)/NDL4 (N4) (EL7047)
//     PlcTask Inputs/MAIN.nott_ics.Delay_Lines.NDL4.i_nCouplerState <-> InfoData/State
//     PlcTask Inputs/MAIN.nott_ics.Delay_Lines.NDL4.switches/bLHW <-> STM Status/Status/Digital input 1
//     PlcTask Inputs/MAIN.nott_ics.Delay_Lines.NDL4.switches/bUHW <-> STM Status/Status/Digital input 2
//   nott_ics/nott_ics Instance <-> Device 1 (EtherCAT)/Term 7 (EK1101)/Term 14 (EK1122)/Term 32 (EK1101)/NTPA1 - NTPA2 (N6) (EL7342)
//     PlcTask Inputs/MAIN.nott_ics.TipTilt.NTPA1.i_nCouplerState <-> InfoData/State
//     PlcTask Inputs/MAIN.nott_ics.TipTilt.NTPA2.i_nCouplerState <-> InfoData/State
//   nott_ics/nott_ics Instance <-> Device 1 (EtherCAT)/Term 7 (EK1101)/Term 14 (EK1122)/Term 32 (EK1101)/NTPA3 - NTPA4 (N7) (EL7342)
//     PlcTask Inputs/MAIN.nott_ics.TipTilt.NTPA3.i_nCouplerState <-> InfoData/State
//     PlcTask Inputs/MAIN.nott_ics.TipTilt.NTPA4.i_nCouplerState <-> InfoData/State
//   nott_ics/nott_ics Instance <-> Device 1 (EtherCAT)/Term 7 (EK1101)/Term 14 (EK1122)/Term 32 (EK1101)/NTPB1 - NTPB2 (N14) (EL7342)
//     PlcTask Inputs/MAIN.nott_ics.TipTilt.NTPB1.i_nCouplerState <-> InfoData/State
//     PlcTask Inputs/MAIN.nott_ics.TipTilt.NTPB2.i_nCouplerState <-> InfoData/State
//   nott_ics/nott_ics Instance <-> Device 1 (EtherCAT)/Term 7 (EK1101)/Term 14 (EK1122)/Term 32 (EK1101)/NTPB3 - NTPB4 (N15) (EL7342)
//     PlcTask Inputs/MAIN.nott_ics.TipTilt.NTPB3.i_nCouplerState <-> InfoData/State
//     PlcTask Inputs/MAIN.nott_ics.TipTilt.NTPB4.i_nCouplerState <-> InfoData/State
//   nott_ics/nott_ics Instance <-> Device 1 (EtherCAT)/Term 7 (EK1101)/Term 14 (EK1122)/Term 32 (EK1101)/NTTA1 - NTTA2 (N9) (EL7342)
//     PlcTask Inputs/MAIN.nott_ics.TipTilt.NTTA1.i_nCouplerState <-> InfoData/State
//     PlcTask Inputs/MAIN.nott_ics.TipTilt.NTTA2.i_nCouplerState <-> InfoData/State
//   nott_ics/nott_ics Instance <-> Device 1 (EtherCAT)/Term 7 (EK1101)/Term 14 (EK1122)/Term 32 (EK1101)/NTTA3 - NTTA4 (N10) (EL7342)
//     PlcTask Inputs/MAIN.nott_ics.TipTilt.NTTA3.i_nCouplerState <-> InfoData/State
//     PlcTask Inputs/MAIN.nott_ics.TipTilt.NTTA4.i_nCouplerState <-> InfoData/State
//   nott_ics/nott_ics Instance <-> Device 1 (EtherCAT)/Term 7 (EK1101)/Term 14 (EK1122)/Term 32 (EK1101)/NTTB1 - NTTB2 (N18) (EL7342)
//     PlcTask Inputs/MAIN.nott_ics.TipTilt.NTTB1.i_nCouplerState <-> InfoData/State
//     PlcTask Inputs/MAIN.nott_ics.TipTilt.NTTB2.i_nCouplerState <-> InfoData/State
//   nott_ics/nott_ics Instance <-> Device 1 (EtherCAT)/Term 7 (EK1101)/Term 14 (EK1122)/Term 32 (EK1101)/NTTB3 - NTTB4 (N19) (EL7342)
//     PlcTask Inputs/MAIN.nott_ics.TipTilt.NTTB3.i_nCouplerState <-> InfoData/State
//     PlcTask Inputs/MAIN.nott_ics.TipTilt.NTTB4.i_nCouplerState <-> InfoData/State
//   nott_ics/nott_ics Instance <-> Device 1 (EtherCAT)/Term 7 (EK1101)/Term 50 (EM3701)
//     PlcTask Inputs/MAIN.nott_ics.CO2_Pressure_Control.nCO2_Diff_Press_Sens <-> AI Inputs/Value
//   nott_ics/nott_ics Instance <-> Device 1 (EtherCAT)/Term 7 (EK1101)/Term 8 (EL2004)
//     PlcTask Inputs/MAIN.nott_ics.CO2_Pressure_Control.CO2_Valve.Actuator.i_nCouplerState <-> InfoData/State
//   nott_ics/nott_ics Instance <-> NC-Task 1 SAF/Axes/NBS
//     PlcTask Inputs/MAIN.nott_ics.Calibration_Unit_Beam_Splitter.NBS.Axis.NcToPlc <-> Outputs/ToPlc
//     PlcTask Outputs/MAIN.nott_ics.Calibration_Unit_Beam_Splitter.NBS.Axis.PlcToNc <-> Inputs/FromPlc
//   nott_ics/nott_ics Instance <-> NC-Task 1 SAF/Axes/NCP1
//     PlcTask Inputs/MAIN.nott_ics.CO2TransStages.NCP1.Axis.NcToPlc <-> Outputs/ToPlc
//     PlcTask Outputs/MAIN.nott_ics.CO2TransStages.NCP1.Axis.PlcToNc <-> Inputs/FromPlc
//   nott_ics/nott_ics Instance <-> NC-Task 1 SAF/Axes/NCP2
//     PlcTask Inputs/MAIN.nott_ics.CO2TransStages.NCP2.Axis.NcToPlc <-> Outputs/ToPlc
//     PlcTask Outputs/MAIN.nott_ics.CO2TransStages.NCP2.Axis.PlcToNc <-> Inputs/FromPlc
//   nott_ics/nott_ics Instance <-> NC-Task 1 SAF/Axes/NCP3
//     PlcTask Inputs/MAIN.nott_ics.CO2TransStages.NCP3.Axis.NcToPlc <-> Outputs/ToPlc
//     PlcTask Outputs/MAIN.nott_ics.CO2TransStages.NCP3.Axis.PlcToNc <-> Inputs/FromPlc
//   nott_ics/nott_ics Instance <-> NC-Task 1 SAF/Axes/NCP4
//     PlcTask Inputs/MAIN.nott_ics.CO2TransStages.NCP4.Axis.NcToPlc <-> Outputs/ToPlc
//     PlcTask Outputs/MAIN.nott_ics.CO2TransStages.NCP4.Axis.PlcToNc <-> Inputs/FromPlc
//   nott_ics/nott_ics Instance <-> NC-Task 1 SAF/Axes/NDL1
//     PlcTask Inputs/MAIN.nott_ics.Delay_Lines.NDL1.Axis.NcToPlc <-> Outputs/ToPlc
//     PlcTask Outputs/MAIN.nott_ics.Delay_Lines.NDL1.Axis.PlcToNc <-> Inputs/FromPlc
//   nott_ics/nott_ics Instance <-> NC-Task 1 SAF/Axes/NDL2
//     PlcTask Inputs/MAIN.nott_ics.Delay_Lines.NDL2.Axis.NcToPlc <-> Outputs/ToPlc
//     PlcTask Outputs/MAIN.nott_ics.Delay_Lines.NDL2.Axis.PlcToNc <-> Inputs/FromPlc
//   nott_ics/nott_ics Instance <-> NC-Task 1 SAF/Axes/NDL3
//     PlcTask Inputs/MAIN.nott_ics.Delay_Lines.NDL3.Axis.NcToPlc <-> Outputs/ToPlc
//     PlcTask Outputs/MAIN.nott_ics.Delay_Lines.NDL3.Axis.PlcToNc <-> Inputs/FromPlc
//   nott_ics/nott_ics Instance <-> NC-Task 1 SAF/Axes/NDL4
//     PlcTask Inputs/MAIN.nott_ics.Delay_Lines.NDL4.Axis.NcToPlc <-> Outputs/ToPlc
//     PlcTask Outputs/MAIN.nott_ics.Delay_Lines.NDL4.Axis.PlcToNc <-> Inputs/FromPlc
//   nott_ics/nott_ics Instance <-> NC-Task 1 SAF/Axes/NGP1
//     PlcTask Inputs/MAIN.nott_ics.ZnSeActuators.NGP1.Axis.NcToPlc <-> Outputs/ToPlc
//     PlcTask Outputs/MAIN.nott_ics.ZnSeActuators.NGP1.Axis.PlcToNc <-> Inputs/FromPlc
//   nott_ics/nott_ics Instance <-> NC-Task 1 SAF/Axes/NGP2
//     PlcTask Inputs/MAIN.nott_ics.ZnSeActuators.NGP2.Axis.NcToPlc <-> Outputs/ToPlc
//     PlcTask Outputs/MAIN.nott_ics.ZnSeActuators.NGP2.Axis.PlcToNc <-> Inputs/FromPlc
//   nott_ics/nott_ics Instance <-> NC-Task 1 SAF/Axes/NGP3
//     PlcTask Inputs/MAIN.nott_ics.ZnSeActuators.NGP3.Axis.NcToPlc <-> Outputs/ToPlc
//     PlcTask Outputs/MAIN.nott_ics.ZnSeActuators.NGP3.Axis.PlcToNc <-> Inputs/FromPlc
//   nott_ics/nott_ics Instance <-> NC-Task 1 SAF/Axes/NGP4
//     PlcTask Inputs/MAIN.nott_ics.ZnSeActuators.NGP4.Axis.NcToPlc <-> Outputs/ToPlc
//     PlcTask Outputs/MAIN.nott_ics.ZnSeActuators.NGP4.Axis.PlcToNc <-> Inputs/FromPlc
//   nott_ics/nott_ics Instance <-> NC-Task 1 SAF/Axes/NPC1
//     PlcTask Inputs/MAIN.nott_ics.Birefringence.NPC1.Axis.NcToPlc <-> Outputs/ToPlc
//     PlcTask Outputs/MAIN.nott_ics.Birefringence.NPC1.Axis.PlcToNc <-> Inputs/FromPlc
//   nott_ics/nott_ics Instance <-> NC-Task 1 SAF/Axes/NPC2
//     PlcTask Inputs/MAIN.nott_ics.Birefringence.NPC2.Axis.NcToPlc <-> Outputs/ToPlc
//     PlcTask Outputs/MAIN.nott_ics.Birefringence.NPC2.Axis.PlcToNc <-> Inputs/FromPlc
//   nott_ics/nott_ics Instance <-> NC-Task 1 SAF/Axes/NPC3
//     PlcTask Inputs/MAIN.nott_ics.Birefringence.NPC3.Axis.NcToPlc <-> Outputs/ToPlc
//     PlcTask Outputs/MAIN.nott_ics.Birefringence.NPC3.Axis.PlcToNc <-> Inputs/FromPlc
//   nott_ics/nott_ics Instance <-> NC-Task 1 SAF/Axes/NPC4
//     PlcTask Inputs/MAIN.nott_ics.Birefringence.NPC4.Axis.NcToPlc <-> Outputs/ToPlc
//     PlcTask Outputs/MAIN.nott_ics.Birefringence.NPC4.Axis.PlcToNc <-> Inputs/FromPlc
//   nott_ics/nott_ics Instance <-> NC-Task 1 SAF/Axes/NSH1
//     PlcTask Inputs/MAIN.nott_ics.Shutters.NSH1.Axis.NcToPlc <-> Outputs/ToPlc
//     PlcTask Outputs/MAIN.nott_ics.Shutters.NSH1.Axis.PlcToNc <-> Inputs/FromPlc
//   nott_ics/nott_ics Instance <-> NC-Task 1 SAF/Axes/NSH2
//     PlcTask Inputs/MAIN.nott_ics.Shutters.NSH2.Axis.NcToPlc <-> Outputs/ToPlc
//     PlcTask Outputs/MAIN.nott_ics.Shutters.NSH2.Axis.PlcToNc <-> Inputs/FromPlc
//   nott_ics/nott_ics Instance <-> NC-Task 1 SAF/Axes/NSH3
//     PlcTask Inputs/MAIN.nott_ics.Shutters.NSH3.Axis.NcToPlc <-> Outputs/ToPlc
//     PlcTask Outputs/MAIN.nott_ics.Shutters.NSH3.Axis.PlcToNc <-> Inputs/FromPlc
//   nott_ics/nott_ics Instance <-> NC-Task 1 SAF/Axes/NSH4
//     PlcTask Inputs/MAIN.nott_ics.Shutters.NSH4.Axis.NcToPlc <-> Outputs/ToPlc
//     PlcTask Outputs/MAIN.nott_ics.Shutters.NSH4.Axis.PlcToNc <-> Inputs/FromPlc
//   nott_ics/nott_ics Instance <-> NC-Task 1 SAF/Axes/NTPA1
//     PlcTask Inputs/MAIN.nott_ics.TipTilt.NTPA1.Axis.NcToPlc <-> Outputs/ToPlc
//     PlcTask Outputs/MAIN.nott_ics.TipTilt.NTPA1.Axis.PlcToNc <-> Inputs/FromPlc
//   nott_ics/nott_ics Instance <-> NC-Task 1 SAF/Axes/NTPA2
//     PlcTask Inputs/MAIN.nott_ics.TipTilt.NTPA2.Axis.NcToPlc <-> Outputs/ToPlc
//     PlcTask Outputs/MAIN.nott_ics.TipTilt.NTPA2.Axis.PlcToNc <-> Inputs/FromPlc
//   nott_ics/nott_ics Instance <-> NC-Task 1 SAF/Axes/NTPA3
//     PlcTask Inputs/MAIN.nott_ics.TipTilt.NTPA3.Axis.NcToPlc <-> Outputs/ToPlc
//     PlcTask Outputs/MAIN.nott_ics.TipTilt.NTPA3.Axis.PlcToNc <-> Inputs/FromPlc
//   nott_ics/nott_ics Instance <-> NC-Task 1 SAF/Axes/NTPA4
//     PlcTask Inputs/MAIN.nott_ics.TipTilt.NTPA4.Axis.NcToPlc <-> Outputs/ToPlc
//     PlcTask Outputs/MAIN.nott_ics.TipTilt.NTPA4.Axis.PlcToNc <-> Inputs/FromPlc
//   nott_ics/nott_ics Instance <-> NC-Task 1 SAF/Axes/NTPB1
//     PlcTask Inputs/MAIN.nott_ics.TipTilt.NTPB1.Axis.NcToPlc <-> Outputs/ToPlc
//     PlcTask Outputs/MAIN.nott_ics.TipTilt.NTPB1.Axis.PlcToNc <-> Inputs/FromPlc
//   nott_ics/nott_ics Instance <-> NC-Task 1 SAF/Axes/NTPB2
//     PlcTask Inputs/MAIN.nott_ics.TipTilt.NTPB2.Axis.NcToPlc <-> Outputs/ToPlc
//     PlcTask Outputs/MAIN.nott_ics.TipTilt.NTPB2.Axis.PlcToNc <-> Inputs/FromPlc
//   nott_ics/nott_ics Instance <-> NC-Task 1 SAF/Axes/NTPB3
//     PlcTask Inputs/MAIN.nott_ics.TipTilt.NTPB3.Axis.NcToPlc <-> Outputs/ToPlc
//     PlcTask Outputs/MAIN.nott_ics.TipTilt.NTPB3.Axis.PlcToNc <-> Inputs/FromPlc
//   nott_ics/nott_ics Instance <-> NC-Task 1 SAF/Axes/NTPB4
//     PlcTask Inputs/MAIN.nott_ics.TipTilt.NTPB4.Axis.NcToPlc <-> Outputs/ToPlc
//     PlcTask Outputs/MAIN.nott_ics.TipTilt.NTPB4.Axis.PlcToNc <-> Inputs/FromPlc
//   nott_ics/nott_ics Instance <-> NC-Task 1 SAF/Axes/NTTA1
//     PlcTask Inputs/MAIN.nott_ics.TipTilt.NTTA1.Axis.NcToPlc <-> Outputs/ToPlc
//     PlcTask Outputs/MAIN.nott_ics.TipTilt.NTTA1.Axis.PlcToNc <-> Inputs/FromPlc
//   nott_ics/nott_ics Instance <-> NC-Task 1 SAF/Axes/NTTA2
//     PlcTask Inputs/MAIN.nott_ics.TipTilt.NTTA2.Axis.NcToPlc <-> Outputs/ToPlc
//     PlcTask Outputs/MAIN.nott_ics.TipTilt.NTTA2.Axis.PlcToNc <-> Inputs/FromPlc
//   nott_ics/nott_ics Instance <-> NC-Task 1 SAF/Axes/NTTA3
//     PlcTask Inputs/MAIN.nott_ics.TipTilt.NTTA3.Axis.NcToPlc <-> Outputs/ToPlc
//     PlcTask Outputs/MAIN.nott_ics.TipTilt.NTTA3.Axis.PlcToNc <-> Inputs/FromPlc
//   nott_ics/nott_ics Instance <-> NC-Task 1 SAF/Axes/NTTA4
//     PlcTask Inputs/MAIN.nott_ics.TipTilt.NTTA4.Axis.NcToPlc <-> Outputs/ToPlc
//     PlcTask Outputs/MAIN.nott_ics.TipTilt.NTTA4.Axis.PlcToNc <-> Inputs/FromPlc
//   nott_ics/nott_ics Instance <-> NC-Task 1 SAF/Axes/NTTB1
//     PlcTask Inputs/MAIN.nott_ics.TipTilt.NTTB1.Axis.NcToPlc <-> Outputs/ToPlc
//     PlcTask Outputs/MAIN.nott_ics.TipTilt.NTTB1.Axis.PlcToNc <-> Inputs/FromPlc
//   nott_ics/nott_ics Instance <-> NC-Task 1 SAF/Axes/NTTB2
//     PlcTask Inputs/MAIN.nott_ics.TipTilt.NTTB2.Axis.NcToPlc <-> Outputs/ToPlc
//     PlcTask Outputs/MAIN.nott_ics.TipTilt.NTTB2.Axis.PlcToNc <-> Inputs/FromPlc
//   nott_ics/nott_ics Instance <-> NC-Task 1 SAF/Axes/NTTB3
//     PlcTask Inputs/MAIN.nott_ics.TipTilt.NTTB3.Axis.NcToPlc <-> Outputs/ToPlc
//     PlcTask Outputs/MAIN.nott_ics.TipTilt.NTTB3.Axis.PlcToNc <-> Inputs/FromPlc
//   nott_ics/nott_ics Instance <-> NC-Task 1 SAF/Axes/NTTB4
//     PlcTask Inputs/MAIN.nott_ics.TipTilt.NTTB4.Axis.NcToPlc <-> Outputs/ToPlc
//     PlcTask Outputs/MAIN.nott_ics.TipTilt.NTTB4.Axis.PlcToNc <-> Inputs/FromPlc
//   nott_ics/nott_ics Instance <-> nott_ics/nott_ics Instance
//     PlcTask Inputs/MAIN.nott_ics.CO2_Pressure_Control.CO2_Valve.Actuator.i_bON <-> PlcTask Outputs/MAIN.nott_ics.CO2_Pressure_Control.CO2_Valve.Actuator.q_bCtrl
//     PlcTask Inputs/MAIN.nott_ics.Calibration_Unit_Beam_Splitter.SIM_NBS.i_bBrake_Ctrl <-> PlcTask Outputs/MAIN.nott_ics.Calibration_Unit_Beam_Splitter.NBS.q_bBrake_Ctrl

CONFIGURATION nott_ics
    RESOURCE PLC ON TwinCAT3
        TASK CameraTrigs(INTERVAL := T#1ms, PRIORITY := 1);
        TASK PlcTask(INTERVAL := T#10ms, PRIORITY := 20);
        TASK VISU_TASK(INTERVAL := T#200000us, PRIORITY := 30);
        PROGRAM INFRATEC_TRIGERS WITH CameraTrigs : INFRATEC_TRIGERS;
        PROGRAM MAIN WITH PlcTask : MAIN;
        PROGRAM PRG_HMI WITH VISU_TASK : PRG_HMI;
    END_RESOURCE
END_CONFIGURATION

// ---- DUTs/Structures/T_NOTT_STAT.TcDUT
TYPE T_NOTT_STAT :
STRUCT

	bEnabled:		BOOL 	:= FALSE;	
	bConfigured:	BOOL	:= FALSE;
	bDone:			BOOL;				// Flag if controller is OK
	bBusy:			BOOL;				// Flag if controller is BUSY
	bError:			BOOL;				// Flag if controller is in ERROR state
	bActive:		BOOL;				// Flag if controller is ACTIVE
	
	sState:			STRING(64);			// State as text
	sError:			STRING(64);			// Error as text
	
	bInterlock:	BOOL := FALSE;			// Flag if any command is prevented
	bWarning:	BOOL := FALSE;			// 
	sStatus:	STRING := 'OK';			// Textual description in case of problems
	
END_STRUCT
END_TYPE

// ---- DUTs/T_NOTT_IR_CAMERA_DL_SYNC.TcDUT
TYPE T_NOTT_IR_CAMERA_DL_SYNC :
STRUCT
	TimeStamp:		ULINT;
	lrActPos_DL1:	LREAL;
	lrActPos_DL2:	LREAL;
	lrActPos_DL3:	LREAL;
	lrActPos_DL4:	LREAL;	
END_STRUCT
END_TYPE

// ---- DUTs/T_NOTT_CAMERA_TIMESTAMPS_N_DL_POS.TcDUT
TYPE T_NOTT_CAMERA_TIMESTAMPS_N_DL_POS :
STRUCT
	TimeStamp:		ULINT;
	lrActPos_DL1:	LREAL;
	lrActPos_DL2:	LREAL;
	lrActPos_DL3:	LREAL;
	lrActPos_DL4:	LREAL;	
END_STRUCT
END_TYPE

// ---- HMI/DUTs/Subsystems/Tip_Tilt/E_HMI_TIP_TILT_TABS.TcDUT
{attribute 'qualified_only'}
{attribute 'strict'}
TYPE E_HMI_TIP_TILT_TABS :
(
	TIP_A,
    TIP_B,
	TILT_A,
    TILT_B

);
END_TYPE

// ---- HMI/DUTs/System/E_HMI_TABS.TcDUT
{attribute 'qualified_only'}
{attribute 'strict'}
TYPE E_HMI_TABS :
(
	HOME,
    SERVICES,
	EVENTS,
	CRYO_INTERLOCKS,
	
	SHUTTERS,
	TIP_TILT,
	DELAY_LINES,
	CO2_TRANSLATION_STAGES,
	ZNSE_ACTUATORS,
	BIREFRINGENCE_ACTUATORS,
	CALIBRATION_UNIT_BEAM_SPLITER,
	CO2_PRESSURE_CONTROL
);
END_TYPE

// ---- HMI/DUTs/Util/E_HMI_COLORS.TcDUT
TYPE E_HMI_COLORS :
(
	GREEN := 16#FF00FF00,
	RED := 16#FFFF0000,
	ORANGE := 16#FFFF802D,
	GRAY := 16#FFD3D3D3,
	DARK_GRAY := 16#FF949494,
	BLACK := 16#FF000000,
	WHITE := 16#FFFFFFFF,
	BLUE := 16#FF0000FF
) DWORD;
END_TYPE

// ---- HMI/DUTs/Util/E_HMI_VOTER_TABS.TcDUT
{attribute 'qualified_only'}
{attribute 'strict'}
TYPE E_HMI_VOTER_TABS :
(
	VOTER_1,
    VOTER_2,
    VOTER_3,
    VOTER_4,
    VOTER_5,
    VOTER_6,
    VOTER_7,
    VOTER_8,
    VOTER_9,
    VOTER_10
);
END_TYPE

// ---- HMI/DUTs/Util/T_ECAT_MODULE.TcDUT
TYPE T_ECAT_MODULE :
STRUCT
    sName : STRING(32);
    sType : STRING(16);
    nState : UINT;
    sState : STRING(16);
    bError : BOOL;
    bDisabled : BOOL;
    bNotPresent : BOOL;
END_STRUCT
END_TYPE

// ---- HMI/DUTs/Util/T_HMI_COLORS.TcDUT
TYPE T_HMI_COLORS :
STRUCT
    fg : E_HMI_COLORS; // foreground
    bg : E_HMI_COLORS; // background
END_STRUCT
END_TYPE

// ---- GVLs/NOTT_GVL.TcGVL
{attribute 'qualified_only'}
VAR_GLOBAL
	// Actual position of the delay lines
	gv_DL1_ActualPos:		LREAL;
	gv_DL2_ActualPos:		LREAL;
	gv_DL3_ActualPos:		LREAL;
	gv_DL4_ActualPos:		LREAL;
	
	
END_VAR

// ---- POUs/Camera_Triggers/INFRATEC_TRIGERS.TcPOU
PROGRAM INFRATEC_TRIGERS
VAR
	
//	Trig_Cam_1 AT %Q*:		BOOL;
//	Trig_Cam_2 AT %Q*:		BOOL;
	
	
//	Cam_response_1 AT %I*:	BOOL;
//	Cam_response_2 AT %I*:	BOOL;
	
//	{attribute 'OPC.UA.DA' := '1'}
//	bTrigCam_1:				BOOL;
//	{attribute 'OPC.UA.DA' := '1'}
//	bTrigCam_2:				BOOL;
	
//	{attribute 'OPC.UA.DA' := '1'}
//	bCamResponse_1:			BOOL;
//	{attribute 'OPC.UA.DA' := '1'}
//	bCamResponse_2:			BOOL;
	
//	Trig1_Sync_Info:		T_NOTT_IR_CAMERA_DL_SYNC;
//	Trig2_Sync_Info:		T_NOTT_IR_CAMERA_DL_SYNC;
	
//	NottTime:			FB_TIME;
	
//	// Time Stamp
//	fbGetSystemTime  : GETSYSTEMTIME;
//	fileTime         : T_FILETIME;
//	{attribute 'OPC.UA.DA':='1'}
//	sPLCTime            : STRING;
	
//	// NTP External Time
	
//	nNTPExternalTime AT %I*: LINT;
//	{attribute 'OPC.UA.DA':='1'}
//	sNTPExtTime:			STRING;
	
END_VAR


//NottTime();



//Trig_Cam_1 := bTrigCam_1;
//Trig_Cam_2 := bTrigCam_2;


//bCamResponse_1 := Cam_response_1;
//bCamResponse_2 := Cam_response_2;

//Trig1_Sync_Info.TimeStamp := NottTime.GetTime();
//Trig1_Sync_Info.lrActPos_DL1 := NOTT_GVL.gv_DL1_ActualPos;
//Trig1_Sync_Info.lrActPos_DL2 := NOTT_GVL.gv_DL1_ActualPos;
//Trig1_Sync_Info.lrActPos_DL3 := NOTT_GVL.gv_DL1_ActualPos;
//Trig1_Sync_Info.lrActPos_DL4 := NOTT_GVL.gv_DL1_ActualPos;

//// Time Stamps

//fbGetSystemTime(timeLoDW=>fileTime.dwLowDateTime, timeHiDW=>fileTime.dwHighDateTime );
//sPLCTime := SYSTEMTIME_TO_STRING( FILETIME_TO_SYSTEMTIME( fileTime ) );

//// NTP External Time

//sNTPExtTime := F_SysTimeToString(nNTPExternalTime);

END_PROGRAM

// ---- POUs/MAIN.TcPOU
PROGRAM MAIN
VAR
	{attribute 'OPC.UA.DA' := '1'}
	nott_ics:		FB_NOTT_ICS;
//	{attribute 'OPC.UA.DA' := '1'}
//	not_cryo_ctrl:	FB_NOTT_CRYO_CTRL;
//	{attribute 'OPC.UA.DA' := '1'}
	fbServices : FB_SERVICES;	
	
END_VAR


nott_ics();

//not_cryo_ctrl();

END_PROGRAM

// ---- POUs/System/FB_NOTT_ICS.TcPOU
FUNCTION_BLOCK FB_NOTT_ICS
VAR_INPUT
END_VAR
VAR_OUTPUT
END_VAR
VAR

	Events:								FB_NOTT_EVENTS;
	Cryo_Interlocks:					FB_NOTT_CRYO_INTERLOCKS;
	
	Shutters:							FB_NOTT_SHUTTERS;
	TipTilt:							FB_NOTT_TIP_TILT;	
	Delay_Lines:						FB_NOTT_DELAY_LINES;
	CO2TransStages:						FB_NOTT_CO2_TRANS_STAGES;
	ZnSeActuators:						FB_NOTT_ZNSE_ACTUATORS;
	Birefringence:						FB_NOTT_BIREFRINGENCE;
	Calibration_Unit_Beam_Splitter:		FB_NOTT_CALIBRATION_BEAM_SPLITTER;
	CO2_Pressure_Control:				FB_NOTT_CO2_PRESSURE_CONTROL;
	
	
END_VAR


Events();
Cryo_Interlocks();

Shutters();
TipTilt();
Delay_Lines();
Delay_Lines.M_SET_DL_ACTUAL_POS();
CO2TransStages();
ZnSeActuators();
Birefringence();
Calibration_Unit_Beam_Splitter();
CO2_Pressure_Control();

END_FUNCTION_BLOCK

// ---- POUs/EVENTS/FB_NOTT_EVENTS.TcPOU
FUNCTION_BLOCK FB_NOTT_EVENTS
VAR_INPUT
END_VAR
VAR_OUTPUT
END_VAR
VAR
END_VAR

END_FUNCTION_BLOCK

// ---- POUs/Cryo_Interlocks/FB_NOTT_CRYO_INTERLOCKS.TcPOU
FUNCTION_BLOCK FB_NOTT_CRYO_INTERLOCKS
VAR_INPUT
END_VAR
VAR_OUTPUT
END_VAR
VAR
		stat:		T_NOTT_STAT;
END_VAR

END_FUNCTION_BLOCK

// ---- POUs/Subsystems/FB_NOTT_SHUTTERS.TcPOU
FUNCTION_BLOCK FB_NOTT_SHUTTERS
VAR_INPUT
END_VAR
VAR_OUTPUT
END_VAR
VAR
	NSH1:		FB_NOTT_MOTOR;
	NSH2:		FB_NOTT_MOTOR;
	NSH3:		FB_NOTT_MOTOR;
	NSH4:		FB_NOTT_MOTOR;
	
	Test_Shutter:	FB_NOTT_MOTOR;
	
	
	ptrShutters:	ARRAY [1..4] OF POINTER TO FB_NOTT_MOTOR;
	// GUI stuff
	guiShutterIndex:	UINT := 1;	// Index for Shutter Engineering GUI
	
	stat:		T_NOTT_STAT;
	
END_VAR



NSH1(
	in_bStepper_Shutter := FALSE,
	in_bSafe:=, 
	in_bDisableIfUnsafe:=, 
	sName:= 'NSH 1', 
	nNOVRAM_DevId:= 6, 
	nNOVRAM_Offset:= 21000);
	
NSH2(
	in_bStepper_Shutter := FALSE,
	in_bSafe:=, 
	in_bDisableIfUnsafe:=, 
	sName:= 'NSH 2', 
	nNOVRAM_DevId:= 6, 
	nNOVRAM_Offset:= 22000);
	
NSH3(
	in_bStepper_Shutter := FALSE,
	in_bSafe:=, 
	in_bDisableIfUnsafe:=, 
	sName:= 'NSH 3', 
	nNOVRAM_DevId:= 6, 
	nNOVRAM_Offset:= 23000);
	
NSH4(
	in_bStepper_Shutter := FALSE,
	in_bSafe:=, 
	in_bDisableIfUnsafe:=, 
	sName:= 'NSH 4', 
	nNOVRAM_DevId:= 6, 
	nNOVRAM_Offset:= 24000);

	
	
M_Configure();


Test_Shutter(
	in_bStepper_Shutter := TRUE,
	in_bSafe:=, 
	in_bDisableIfUnsafe:=, 
	sName:= 'Test Shutter', 
	nNOVRAM_DevId:= 6, 
	nNOVRAM_Offset:= 50000);

METHOD M_Configure : BOOL
VAR_INPUT
END_VAR

ptrShutters[1] := ADR(NSH1);
ptrShutters[2] := ADR(NSH2);
ptrShutters[3] := ADR(NSH3);
ptrShutters[4] := ADR(NSH4);
END_METHOD

END_FUNCTION_BLOCK

// ---- POUs/Devices/NOTT_Motor/FB_NOTT_MOTOR.TcPOU
FUNCTION_BLOCK FB_NOTT_MOTOR EXTENDS FB_MOTOR
VAR_INPUT
	in_bStepper_Shutter:	BOOL := FALSE;
END_VAR
VAR_OUTPUT
END_VAR
VAR
	bShutterPartiallyOpen: BOOL := FALSE;
END_VAR


M_CheckShutterStatus();

SUPER^();

METHOD M_CheckShutterStatus
VAR_INPUT
END_VAR

bShutterPartiallyOpen := NOT (stat.signals[0].bActive OR stat.signals[5].bActive);
END_METHOD

{attribute 'TcRpcEnable':='1'}
METHOD RPC_CloseShutter : INT
VAR
	lrVel:	LREAL := 15.0;
END_VAR
IF NOT in_bStepper_Shutter THEN
	RPC_CloseShutter	:= M_SetRpcStatus(E_MOTOR_RPC_ERROR.UNSAFE);
	RETURN;
END_IF

// If unsafe, move is not allowed.
IF NOT in_bSafe THEN
	RPC_CloseShutter	:= M_SetRpcStatus(E_MOTOR_RPC_ERROR.UNSAFE);
	RETURN;
END_IF

// RPC calls are not allowed in Local mode.
IF stat.bLocal THEN
	RPC_CloseShutter	:= M_SetRpcStatus(E_MOTOR_RPC_ERROR.LOCAL);
	RETURN;
END_IF

// Move in Velocity command is accepted only in OP state.
IF	stat.nState <> E_MOTOR_STATE.OP	THEN
	RPC_CloseShutter	:= M_SetRpcStatus(E_MOTOR_RPC_ERROR.NOT_OP);
	RETURN;
// Set velocity cannot be 0.0.
ELSIF	lrVel = 0.0	THEN
	RPC_CloseShutter	:= M_SetRpcStatus(E_MOTOR_RPC_ERROR.VEL_ZERO);
	RETURN;
// Set velocity cannot be greater than MAX Velocity.
// Note that MoveVel() accepts negative velocity. That is
// why we use ABS().
ELSIF	ABS(lrVel) > stat.axis.lrMaxVelocity	THEN
	RPC_CloseShutter	:= M_SetRpcStatus(E_MOTOR_RPC_ERROR.VEL_MAX);
	RETURN;
ELSE
	// Set command
	ctrl.nCommand 		:= E_MOTOR_COMMAND.MOTOR_MOVE;
	ctrl.nMoveType		:= E_MOTOR_MOVE_TYPE.VELOCITY;

	ctrl.lrVelocity		:= lrVel;
	ctrl.nDirection		:= MC_Positive_Direction;


	ctrl.bExecute 		:= TRUE;
	
	// Call was successful
	RPC_CloseShutter	:= M_SetRpcStatus(E_MOTOR_RPC_ERROR.OK);
END_IF
END_METHOD

{attribute 'TcRpcEnable':='1'}
METHOD RPC_OpenShutter : INT
VAR
	lrVel:	LREAL := 15.0;
END_VAR
IF NOT in_bStepper_Shutter THEN
	RPC_OpenShutter	:= M_SetRpcStatus(E_MOTOR_RPC_ERROR.UNSAFE);
	RETURN;
END_IF

// If unsafe, move is not allowed.
IF NOT in_bSafe THEN
	RPC_OpenShutter	:= M_SetRpcStatus(E_MOTOR_RPC_ERROR.UNSAFE);
	RETURN;
END_IF

// RPC calls are not allowed in Local mode.
IF stat.bLocal THEN
	RPC_OpenShutter	:= M_SetRpcStatus(E_MOTOR_RPC_ERROR.LOCAL);
	RETURN;
END_IF

// Move in Velocity command is accepted only in OP state.
IF	stat.nState <> E_MOTOR_STATE.OP	THEN
	RPC_OpenShutter	:= M_SetRpcStatus(E_MOTOR_RPC_ERROR.NOT_OP);
	RETURN;
// Set velocity cannot be 0.0.
ELSIF	lrVel = 0.0	THEN
	RPC_OpenShutter	:= M_SetRpcStatus(E_MOTOR_RPC_ERROR.VEL_ZERO);
	RETURN;
// Set velocity cannot be greater than MAX Velocity.
// Note that MoveVel() accepts negative velocity. That is
// why we use ABS().
ELSIF	ABS(lrVel) > stat.axis.lrMaxVelocity	THEN
	RPC_OpenShutter	:= M_SetRpcStatus(E_MOTOR_RPC_ERROR.VEL_MAX);
	RETURN;
ELSE
	// Set command
	ctrl.nCommand 		:= E_MOTOR_COMMAND.MOTOR_MOVE;
	ctrl.nMoveType		:= E_MOTOR_MOVE_TYPE.VELOCITY;

	ctrl.lrVelocity		:= lrVel;
	ctrl.nDirection		:= MC_Negative_Direction;


	ctrl.bExecute 		:= TRUE;
	
	// Call was successful
	RPC_OpenShutter	:= M_SetRpcStatus(E_MOTOR_RPC_ERROR.OK);
END_IF
END_METHOD

END_FUNCTION_BLOCK

// ---- POUs/Subsystems/FB_NOTT_TIP_TILT.TcPOU
FUNCTION_BLOCK FB_NOTT_TIP_TILT
VAR
	
	stat:		T_NOTT_STAT;
	
//	Tip Actuators A 

	NTPA1:			FB_NOTT_MOTOR;
	NTPA2:			FB_NOTT_MOTOR;
	NTPA3:			FB_NOTT_MOTOR;
	NTPA4:			FB_NOTT_MOTOR;
	
	ptrTipActuatorsA:	ARRAY [1..4] OF POINTER TO FB_NOTT_MOTOR;
	// GUI stuff
	guiTipActuatorsAIndex:	UINT := 1;	// Index for Tip Actuators A Engineering GUI

//	Tilt Actuators A 
	
	NTTA1:			FB_NOTT_MOTOR;
	NTTA2:			FB_NOTT_MOTOR;
	NTTA3:			FB_NOTT_MOTOR;
	NTTA4:			FB_NOTT_MOTOR;
	
	ptrTiltActuatorsA:	ARRAY [1..4] OF POINTER TO FB_NOTT_MOTOR;
	// GUI stuff
	guiTiltActuatorsAIndex:	UINT := 1;	// Index for Tilt Actuators A Engineering GUI	
	
//	Tip Actuators B 

	NTPB1:			FB_NOTT_MOTOR;
	NTPB2:			FB_NOTT_MOTOR;
	NTPB3:			FB_NOTT_MOTOR;
	NTPB4:			FB_NOTT_MOTOR;
	
	ptrTipActuatorsB:	ARRAY [1..4] OF POINTER TO FB_NOTT_MOTOR;
	// GUI stuff
	guiTipActuatorsBIndex:	UINT := 1;	// Index for Tip Actuators B Engineering GUI	

//	Tilt Actuators B 
	
	NTTB1:			FB_NOTT_MOTOR;
	NTTB2:			FB_NOTT_MOTOR;
	NTTB3:			FB_NOTT_MOTOR;
	NTTB4:			FB_NOTT_MOTOR;
	
	ptrTiltActuatorsB:	ARRAY [1..4] OF POINTER TO FB_NOTT_MOTOR;
	// GUI stuff
	guiTiltActuatorsBIndex:	UINT := 1;	// Index for Tilt Actuators A Engineering GUI

// Simulation

//	Sim Tip Actuators A 

	SIM_NTPA1:			FB_SIM_MOTOR;
	SIM_NTPA2:			FB_SIM_MOTOR;
	SIM_NTPA3:			FB_SIM_MOTOR;
	SIM_NTPA4:			FB_SIM_MOTOR;

//	Sim Tilt Actuators A 
	
	SIM_NTTA1:			FB_SIM_MOTOR;
	SIM_NTTA2:			FB_SIM_MOTOR;
	SIM_NTTA3:			FB_SIM_MOTOR;
	SIM_NTTA4:			FB_SIM_MOTOR;
	
//	Sim Tip Actuators B 

	SIM_NTPB1:			FB_SIM_MOTOR;
	SIM_NTPB2:			FB_SIM_MOTOR;
	SIM_NTPB3:			FB_SIM_MOTOR;
	SIM_NTPB4:			FB_SIM_MOTOR;
		

//	Sim Tilt Actuators B 
	
	SIM_NTTB1:			FB_SIM_MOTOR;
	SIM_NTTB2:			FB_SIM_MOTOR;
	SIM_NTTB3:			FB_SIM_MOTOR;
	SIM_NTTB4:			FB_SIM_MOTOR;	
	
END_VAR

M_Configure();

//	Tip Actuators A 

NTPA1(
	in_bSafe:= , 
	in_bDisableIfUnsafe:= , 
	sName:= 'NTPA 1', 
	nNOVRAM_DevId:= 6, 
	nNOVRAM_Offset:= 5000);
	
NTPA2(
	in_bSafe:= , 
	in_bDisableIfUnsafe:= , 
	sName:= 'NTPA 2', 
	nNOVRAM_DevId:= 6, 
	nNOVRAM_Offset:= 6000);
	
NTPA3(
	in_bSafe:= , 
	in_bDisableIfUnsafe:= , 
	sName:= 'NTPA 3', 
	nNOVRAM_DevId:= 6, 
	nNOVRAM_Offset:= 7000);
	
NTPA4(
	in_bSafe:= , 
	in_bDisableIfUnsafe:= , 
	sName:= 'NTPA 4', 
	nNOVRAM_DevId:= 6, 
	nNOVRAM_Offset:= 8000);
	
//	Tilt Actuators A
	
NTTA1(
	in_bSafe:= , 
	in_bDisableIfUnsafe:= , 
	sName:= 'NTTA 1', 
	nNOVRAM_DevId:= 6, 
	nNOVRAM_Offset:= 9000);
	
NTTA2(
	in_bSafe:= , 
	in_bDisableIfUnsafe:= , 
	sName:= 'NTTA 2', 
	nNOVRAM_DevId:= 6, 
	nNOVRAM_Offset:= 10000);
	
NTTA3(
	in_bSafe:= , 
	in_bDisableIfUnsafe:= , 
	sName:= 'NTTA 3', 
	nNOVRAM_DevId:= 6, 
	nNOVRAM_Offset:= 11000);
	
NTTA4(
	in_bSafe:= , 
	in_bDisableIfUnsafe:= , 
	sName:= 'NTTA 4', 
	nNOVRAM_DevId:= 6, 
	nNOVRAM_Offset:= 12000);
	
//	Tip Actuators B

NTPB1(
	in_bSafe:= , 
	in_bDisableIfUnsafe:= , 
	sName:= 'NTPB 1', 
	nNOVRAM_DevId:= 6, 
	nNOVRAM_Offset:= 13000);
	
NTPB2(
	in_bSafe:= , 
	in_bDisableIfUnsafe:= , 
	sName:= 'NTPB 2', 
	nNOVRAM_DevId:= 6, 
	nNOVRAM_Offset:= 14000);
	
NTPB3(
	in_bSafe:= , 
	in_bDisableIfUnsafe:= , 
	sName:= 'NTPB 3', 
	nNOVRAM_DevId:= 6, 
	nNOVRAM_Offset:= 15000);
	
NTPB4(
	in_bSafe:= , 
	in_bDisableIfUnsafe:= , 
	sName:= 'NTPB 4', 
	nNOVRAM_DevId:= 6, 
	nNOVRAM_Offset:= 16000);

//	Tilt Actuators B 

NTTB1(
	in_bSafe:= , 
	in_bDisableIfUnsafe:= , 
	sName:= 'NTTB 1', 
	nNOVRAM_DevId:= 6, 
	nNOVRAM_Offset:= 17000);
	
NTTB2(
	in_bSafe:= , 
	in_bDisableIfUnsafe:= , 
	sName:= 'NTTB 2', 
	nNOVRAM_DevId:= 6, 
	nNOVRAM_Offset:= 18000);
	
NTTB3(
	in_bSafe:= , 
	in_bDisableIfUnsafe:= , 
	sName:= 'NTTB 3', 
	nNOVRAM_DevId:= 6, 
	nNOVRAM_Offset:= 19000);
	
NTTB4(
	in_bSafe:= , 
	in_bDisableIfUnsafe:= , 
	sName:= 'NTTB 4', 
	nNOVRAM_DevId:= 6, 
	nNOVRAM_Offset:= 20000);

// Simulation

SIM_NTPA1(ptrCfg:= ADR(NTPA1.cfg), ptrStat:= ADR(NTPA1.stat));
SIM_NTPA2(ptrCfg:= ADR(NTPA2.cfg), ptrStat:= ADR(NTPA2.stat));
SIM_NTPA3(ptrCfg:= ADR(NTPA3.cfg), ptrStat:= ADR(NTPA3.stat));
SIM_NTPA4(ptrCfg:= ADR(NTPA4.cfg), ptrStat:= ADR(NTPA4.stat));

SIM_NTPB1(ptrCfg:= ADR(NTPB1.cfg), ptrStat:= ADR(NTPB1.stat));
SIM_NTPB2(ptrCfg:= ADR(NTPB2.cfg), ptrStat:= ADR(NTPB2.stat));
SIM_NTPB3(ptrCfg:= ADR(NTPB3.cfg), ptrStat:= ADR(NTPB3.stat));
SIM_NTPB4(ptrCfg:= ADR(NTPB4.cfg), ptrStat:= ADR(NTPB4.stat));

SIM_NTTA1(ptrCfg:= ADR(NTTA1.cfg), ptrStat:= ADR(NTTA1.stat));
SIM_NTTA2(ptrCfg:= ADR(NTTA2.cfg), ptrStat:= ADR(NTTA2.stat));
SIM_NTTA3(ptrCfg:= ADR(NTTA3.cfg), ptrStat:= ADR(NTTA3.stat));
SIM_NTTA4(ptrCfg:= ADR(NTTA4.cfg), ptrStat:= ADR(NTTA4.stat));

SIM_NTTB1(ptrCfg:= ADR(NTTB1.cfg), ptrStat:= ADR(NTTB1.stat));
SIM_NTTB2(ptrCfg:= ADR(NTTB2.cfg), ptrStat:= ADR(NTTB2.stat));
SIM_NTTB3(ptrCfg:= ADR(NTTB3.cfg), ptrStat:= ADR(NTTB3.stat));
SIM_NTTB4(ptrCfg:= ADR(NTTB4.cfg), ptrStat:= ADR(NTTB4.stat));

METHOD M_Configure : BOOL
VAR_INPUT
END_VAR
//	Tip Actuators A 

ptrTipActuatorsA[1] := ADR(NTPA1);
ptrTipActuatorsA[2] := ADR(NTPA2);
ptrTipActuatorsA[3] := ADR(NTPA3);
ptrTipActuatorsA[4] := ADR(NTPA4);

//	Tilt Actuators A 

ptrTiltActuatorsA[1] := ADR(NTTA1);
ptrTiltActuatorsA[2] := ADR(NTTA2);
ptrTiltActuatorsA[3] := ADR(NTTA3);
ptrTiltActuatorsA[4] := ADR(NTTA4);

//	Tip Actuators B

ptrTipActuatorsB[1] := ADR(NTPB1);
ptrTipActuatorsB[2] := ADR(NTPB2);
ptrTipActuatorsB[3] := ADR(NTPB3);
ptrTipActuatorsB[4] := ADR(NTPB4);

//	Tilt Actuators B

ptrTiltActuatorsB[1] := ADR(NTTB1);
ptrTiltActuatorsB[2] := ADR(NTTB2);
ptrTiltActuatorsB[3] := ADR(NTTB3);
ptrTiltActuatorsB[4] := ADR(NTTB4);
END_METHOD

END_FUNCTION_BLOCK

// ---- POUs/Subsystems/FB_NOTT_DELAY_LINES.TcPOU
FUNCTION_BLOCK FB_NOTT_DELAY_LINES
VAR_INPUT
END_VAR
VAR_OUTPUT
END_VAR
VAR
	NDL1:		FB_NOTT_MOTOR;
	NDL2:		FB_NOTT_MOTOR;
	NDL3:		FB_NOTT_MOTOR;
	NDL4:		FB_NOTT_MOTOR;
	
	ptrDelayLines:	ARRAY [1..4] OF POINTER TO FB_NOTT_MOTOR;
	// GUI stuff
	guiDLIndex:	UINT := 1;	// Index for Shutter Engineering GUI
	
	stat:		T_NOTT_STAT;
END_VAR

NDL1(
	in_bSafe:=, 
	in_bDisableIfUnsafe:=, 
	sName:= 'NDL 1', 
	nNOVRAM_DevId:= 6, 
	nNOVRAM_Offset:= 1000);
	
NDL2(
	in_bSafe:=, 
	in_bDisableIfUnsafe:=, 
	sName:= 'NDL 2', 
	nNOVRAM_DevId:= 6, 
	nNOVRAM_Offset:= 2000);
	
NDL3(
	in_bSafe:=, 
	in_bDisableIfUnsafe:=, 
	sName:= 'NDL 3', 
	nNOVRAM_DevId:= 6, 
	nNOVRAM_Offset:= 3000);
	
NDL4(
	in_bSafe:=, 
	in_bDisableIfUnsafe:=, 
	sName:= 'NDL 4', 
	nNOVRAM_DevId:= 6, 
	nNOVRAM_Offset:= 4000);
	

M_Configure();

METHOD M_Configure : BOOL
VAR_INPUT
END_VAR

ptrDelayLines[1] := ADR(NDL1);
ptrDelayLines[2] := ADR(NDL2);
ptrDelayLines[3] := ADR(NDL3);
ptrDelayLines[4] := ADR(NDL4);
END_METHOD

METHOD M_SET_DL_ACTUAL_POS : BOOL
VAR_INPUT
END_VAR

NOTT_GVL.gv_DL1_ActualPos := NDL1.M_GetActualPos();
NOTT_GVL.gv_DL2_ActualPos := NDL2.M_GetActualPos();
NOTT_GVL.gv_DL3_ActualPos := NDL3.M_GetActualPos();
NOTT_GVL.gv_DL4_ActualPos := NDL4.M_GetActualPos();
END_METHOD

END_FUNCTION_BLOCK

// ---- POUs/Subsystems/FB_NOTT_CO2_TRANS_STAGES.TcPOU
FUNCTION_BLOCK FB_NOTT_CO2_TRANS_STAGES
VAR_INPUT
END_VAR
VAR_OUTPUT
END_VAR
VAR
	NCP1:		FB_NOTT_MOTOR;
	NCP2:		FB_NOTT_MOTOR;
	NCP3:		FB_NOTT_MOTOR;
	NCP4:		FB_NOTT_MOTOR;
	
	
	ptrNCPs:	ARRAY [1..4] OF POINTER TO FB_NOTT_MOTOR;
	// GUI stuff
	guiNCPsIndex:	UINT := 1;	// Index for Shutter Engineering GUI
	
	stat:		T_NOTT_STAT;
	
END_VAR



NCP1(
	in_bSafe:=, 
	in_bDisableIfUnsafe:=, 
	sName:= 'NCP 1', 
	nNOVRAM_DevId:= 6, 
	nNOVRAM_Offset:= 25000);
	
NCP2(
	in_bSafe:=, 
	in_bDisableIfUnsafe:=, 
	sName:= 'NCP 2', 
	nNOVRAM_DevId:= 6, 
	nNOVRAM_Offset:= 26000);
	
NCP3(
	in_bSafe:=, 
	in_bDisableIfUnsafe:=, 
	sName:= 'NCP 3', 
	nNOVRAM_DevId:= 6, 
	nNOVRAM_Offset:= 27000);
	
NCP4(
	in_bSafe:=, 
	in_bDisableIfUnsafe:=, 
	sName:= 'NCP 4', 
	nNOVRAM_DevId:= 6, 
	nNOVRAM_Offset:= 28000);

	
M_Configure();

METHOD M_Configure : BOOL
VAR_INPUT
END_VAR

ptrNCPs[1] := ADR(NCP1);
ptrNCPs[2] := ADR(NCP2);
ptrNCPs[3] := ADR(NCP3);
ptrNCPs[4] := ADR(NCP4);
END_METHOD

END_FUNCTION_BLOCK

// ---- POUs/Subsystems/FB_NOTT_ZNSE_ACTUATORS.TcPOU
FUNCTION_BLOCK FB_NOTT_ZNSE_ACTUATORS
VAR_INPUT
END_VAR
VAR_OUTPUT
END_VAR
VAR
	NGP1:		FB_NOTT_MOTOR;
	NGP2:		FB_NOTT_MOTOR;
	NGP3:		FB_NOTT_MOTOR;
	NGP4:		FB_NOTT_MOTOR;
	
	
	ptrNGPs:	ARRAY [1..4] OF POINTER TO FB_NOTT_MOTOR;
	// GUI stuff
	guiNGPsIndex:	UINT := 1;	// Index for Shutter Engineering GUI
	
	stat:		T_NOTT_STAT;
	
END_VAR



NGP1(
	in_bSafe:=, 
	in_bDisableIfUnsafe:=, 
	sName:= 'NGP 1', 
	nNOVRAM_DevId:= 6, 
	nNOVRAM_Offset:= 29000);
	
NGP2(
	in_bSafe:=, 
	in_bDisableIfUnsafe:=, 
	sName:= 'NGP 2', 
	nNOVRAM_DevId:= 6, 
	nNOVRAM_Offset:= 30000);
	
NGP3(
	in_bSafe:=, 
	in_bDisableIfUnsafe:=, 
	sName:= 'NGP 3', 
	nNOVRAM_DevId:= 6, 
	nNOVRAM_Offset:= 31000);
	
NGP4(
	in_bSafe:=, 
	in_bDisableIfUnsafe:=, 
	sName:= 'NGP 4', 
	nNOVRAM_DevId:= 6, 
	nNOVRAM_Offset:= 32000);

	
M_Configure();

METHOD M_Configure : BOOL
VAR_INPUT
END_VAR

ptrNGPs[1] := ADR(NGP1);
ptrNGPs[2] := ADR(NGP2);
ptrNGPs[3] := ADR(NGP3);
ptrNGPs[4] := ADR(NGP4);
END_METHOD

END_FUNCTION_BLOCK

// ---- POUs/Subsystems/FB_NOTT_BIREFRINGENCE.TcPOU
FUNCTION_BLOCK FB_NOTT_BIREFRINGENCE
VAR_INPUT
END_VAR
VAR_OUTPUT
END_VAR
VAR
	NPC1:		FB_NOTT_MOTOR;
	NPC2:		FB_NOTT_MOTOR;
	NPC3:		FB_NOTT_MOTOR;
	NPC4:		FB_NOTT_MOTOR;
	
	
	ptrNPCs:	ARRAY [1..4] OF POINTER TO FB_NOTT_MOTOR;
	// GUI stuff
	guiNPCsIndex:	UINT := 1;	// Index for Shutter Engineering GUI
	
	stat:		T_NOTT_STAT;
	
END_VAR



NPC1(
	in_bSafe:=, 
	in_bDisableIfUnsafe:=, 
	sName:= 'NPC 1', 
	nNOVRAM_DevId:= 6, 
	nNOVRAM_Offset:= 33000);
	
NPC2(
	in_bSafe:=, 
	in_bDisableIfUnsafe:=, 
	sName:= 'NPC 2', 
	nNOVRAM_DevId:= 6, 
	nNOVRAM_Offset:= 34000);
	
NPC3(
	in_bSafe:=, 
	in_bDisableIfUnsafe:=, 
	sName:= 'NPC 3', 
	nNOVRAM_DevId:= 6, 
	nNOVRAM_Offset:= 35000);
	
NPC4(
	in_bSafe:=, 
	in_bDisableIfUnsafe:=, 
	sName:= 'NPC 4', 
	nNOVRAM_DevId:= 6, 
	nNOVRAM_Offset:= 36000);

	
M_Configure();

METHOD M_Configure : BOOL
VAR_INPUT
END_VAR

ptrNPCs[1] := ADR(NPC1);
ptrNPCs[2] := ADR(NPC2);
ptrNPCs[3] := ADR(NPC3);
ptrNPCs[4] := ADR(NPC4);
END_METHOD

END_FUNCTION_BLOCK

// ---- POUs/Subsystems/FB_NOTT_CALIBRATION_BEAM_SPLITTER.TcPOU
FUNCTION_BLOCK FB_NOTT_CALIBRATION_BEAM_SPLITTER
VAR_INPUT
END_VAR
VAR_OUTPUT
END_VAR
VAR
	NBS:		FB_NOTT_MOTOR;
	
	SIM_NBS:	FB_SIM_MOTOR;
	
	stat:		T_NOTT_STAT;
END_VAR



NBS(
	in_bSafe:=, 
	in_bDisableIfUnsafe:=, 
	sName:= 'NBS', 
	nNOVRAM_DevId:= 6, 
	nNOVRAM_Offset:= 37000);
	
SIM_NBS (ptrCfg:=ADR(NBS.cfg), ptrStat:=ADR(NBS.stat));

END_FUNCTION_BLOCK

// ---- POUs/Subsystems/FB_NOTT_CO2_PRESSURE_CONTROL.TcPOU
FUNCTION_BLOCK FB_NOTT_CO2_PRESSURE_CONTROL
VAR_INPUT
END_VAR
VAR_OUTPUT
END_VAR
VAR
	CO2_Valve:	FB_CRYO_VALVE_CTRL;
	
	// Pointers to valves
	ptrV:	 POINTER TO FB_CRYO_VALVE_CTRL;
	// Pointers to valve commands
	ptrVC:	 POINTER TO FB_CRYO_CMD_OVERRIDE;
	// Pointers to Enable flags for valves
	ptrEV:	 POINTER TO BOOL;
	
	cor_CO2_Valve:	FB_CRYO_CMD_OVERRIDE;
	bEnable_CO2_Valve:	BOOL := FALSE;
		
	
	
	stat:		T_NOTT_STAT;
	
	nCO2_Diff_Press_Sens AT %I*	:INT;
	lrCO2_Diff_Press_mbar:		LREAL;
	
	bConfigured:		BOOL := FALSE;
	
END_VAR



M_Configure();

M_ReadSensors();

M_Execute_Controller();

METHOD M_Configure : BOOL
VAR_INPUT
END_VAR


IF NOT bConfigured THEN




	ptrV := ADR(CO2_Valve);
	
	
	// Set pointers to Valve Commands - MUST!!!
	ptrVC	:= ADR(cor_CO2_Valve);
	
	ptrEV	:= ADR(bEnable_CO2_Valve);
	
	
	
	
	bConfigured := TRUE;


END_IF
END_METHOD

METHOD M_Execute_Controller : BOOL
VAR_INPUT
END_VAR
cor_CO2_Valve(in_bEnable := bEnable_CO2_Valve);	// Handling of PVV1 commands

CO2_Valve(
	in_sName			:= 'CO2_Valve', 
	in_bEnable			:= cor_CO2_Valve.out_bEnable,
	in_nFeedback		:= E_CRYO_BIN_ACT_FEEDBACK.ON_ONLY);
END_METHOD

METHOD M_ReadSensors : BOOL
VAR_INPUT
END_VAR


lrCO2_Diff_Press_mbar := nCO2_Diff_Press_Sens * 0.01;
END_METHOD

END_FUNCTION_BLOCK

// ---- POUs/Valve/FB_CRYO_VALVE_CTRL.TcPOU
FUNCTION_BLOCK FB_CRYO_VALVE_CTRL EXTENDS FB_CRYO_BIN_CTRL
VAR_INPUT
END_VAR
VAR_OUTPUT
END_VAR
VAR
	//
	// Alarm handling
	//
	// List of alarms to be handled by Valve.
	// Alarms cannot be defined in FB_CRYO_BIN_CTRL,
	// because they are specific to the device/controller.
	// There are three alarms for Valves:
	//   0: NOT_OP
	//   1: CLOSE failed
	//   2: OPEN  failed
	arrEventEntry : ARRAY [0..2] OF TcEventEntry;
	// Alarm handler FB
	fbAlarmHandler : FB_AlarmHandler;
END_VAR

// This call just configures logs at the very start.
// Logging is done by explicit calls to M_LogInfo().
logs(in_sName := in_sName);


// Execute parent FB.
SUPER^();


// Update the status.
// This will handle alarms as well.
M_SetStatus(stat.nState);

METHOD M_Configure
VAR_INPUT
END_VAR
// Device specific implementation
// 
arrEventEntry[0] := Tc_Events.CryoValveEventClass.HardwareError;
arrEventEntry[1] := Tc_Events.CryoValveEventClass.FailureOpen;
arrEventEntry[2] := Tc_Events.CryoValveEventClass.FailureClose;


// A MUST !!!
stat.bConfigured	:= TRUE;
END_METHOD

//
// Overrides the same method in FB_CRYO_BIN_CTRL.
//
// Set labels for logging.
//	OPEN, CLOSE (for valves)
METHOD M_GetStateLabel : STRING
VAR_INPUT
	state:	E_CRYO_BIN_CTRL_STATE;
END_VAR
CASE state OF
	E_CRYO_BIN_CTRL_STATE.OFF:
		M_GetStateLabel	:= 'CLOSED';
	
	E_CRYO_BIN_CTRL_STATE.ACTIVE_SWITCHING_ON:
		M_GetStateLabel	:= 'OPENING...';
	
	E_CRYO_BIN_CTRL_STATE.ACTIVE_OFF:
		M_GetStateLabel	:= 'CLOSED';
	
	E_CRYO_BIN_CTRL_STATE.ACTIVE_ON:
		M_GetStateLabel	:= 'OPEN';
	
